// TIA Portal project "HydroelectricDam Project" (V15)

(* hardware
DEVICE "S71500/ET200MP station_1"  S7-1500 station
   slot 0: "Rail_0"  Rack  6ES7 590-1***0-0AA0
   slot 1: "PLC_1"  CPU 1511-1 PN  6ES7 511-1AK00-0AB0  V1.8
      slot 3: "CPU display_1"  6ES7591-1AA00-0AA0
DEVICE "PC-System_1"  SIMATIC PC station
   slot 0: "SIMATIC PC station"  Rail  SIMATIC PC-Station  V1.0
      slot 125: "Stationmanager"  Station_Manager  V6.0.4
   slot 1: "HMI_RT_1"  WinCC RT Advanced  6AV2 104-0xxxx-xxxx  15.0.0.0
      slot 33792: "Host interface"  Host interface
   slot 2: "IE general_1"  IE General  IE_CP  V8.2.0
*)

// ===== PLC "PLC_1"  CPU 1511-1 PN =====

VAR_GLOBAL   // PLC tag table "Default tag table"
   "Brake_Out" AT %M0.0 : Bool;
   "Baffle_Out" AT %MW18 : Int;
   "RPM_In" AT %MW2 : Int;
   "OilTemp_In" AT %MW4 : Int;
   "Baffle_En" AT %M0.1 : Bool;
   "Current_In" AT %MW6 : Int;
   "OilPumpVFDsp_Out" AT %MW8 : Int;
   "OilPumpVFDen_Out" AT %M0.2 : Bool;
   "OilFlow_In" AT %MW10 : Int;
   "PB_LAD" AT %M0.3 : Bool;
   "ONS" AT %M0.4 : Bool;
   "ProgLang" AT %MW12 : Int;
   "PB_FBD" AT %M0.5 : Bool;
   "PB_SCL" AT %M0.6 : Bool;
   "PB_STL" AT %M0.7 : Bool;
   "ONS1" AT %M1.0 : Bool;
   "ONS2" AT %M1.1 : Bool;
   "ONS3" AT %M1.2 : Bool;
   "AlarmHorn_Out" AT %M1.3 : Bool;
   "StationInterlock_Out" AT %M1.4 : Bool;
   "OilPump_VFD_Pct" AT %MW14 : Int;
   "Baffle_Pct" AT %MW16 : Int;
   "OilTemp" AT %MW20 : Int;
   "OilFlow" AT %MW22 : Int;
   "RPM" AT %MW24 : Int;
   "Current" AT %MW26 : Int;
   "SimLogicEn" AT %M1.5 : Bool;
   "OilPumpVFD_Off_Pb" AT %M1.6 : Bool;
   "OilPumpVFD_Hand_Pb" AT %M1.7 : Bool;
   "OilPumpVFD_Auto_Pb" AT %M30.0 : Bool;
   "Brake_Off_Pb" AT %M30.1 : Bool;
   "Brake_hand_Pb" AT %M30.2 : Bool;
   "Brake_Auto_Pb" AT %M30.3 : Bool;
   "Brake_HOA" AT %MW32 : Int;
   "AlarmHorn_Off_Pb" AT %M30.4 : Bool;
   "AlarmHorn_Hand_Pb" AT %M30.5 : Bool;
   "AlarmHorn_Auto_Pb" AT %M30.6 : Bool;
   "AlarmHorn_HOA" AT %MW34 : Int;
   "StationInterlock_Off_Pb" AT %M30.7 : Bool;
   "StationInterlock_Hand_Pb" AT %M31.0 : Bool;
   "StationInterlock_Auto_Pb" AT %M31.1 : Bool;
   "StationInterlock_HOA" AT %MW36 : Int;
   "OilPumpVFD_Ctrl" AT %M31.2 : Bool;
   "Brake_Ctrl" AT %M31.3 : Bool;
   "Alarm_Horn_Ctrl" AT %M31.4 : Bool;
   "StationInterlock_Ctrl" AT %M31.5 : Bool;
   "AlarmReset" AT %M31.6 : Bool;
   "AlarmSilence" AT %M31.7 : Bool;
   "OilLowFlowAlarm" AT %M42.0 : Bool;
   "OilLowFlowNotify" AT %M42.1 : Bool;
   "OilLowFlow_Sp" AT %MW44 : Int;
   "OvercurrentDelaySpt" AT %MW46 : Int;
   "Overcurrent_Sp" AT %MW48 : Int;
   "OvercurrentAlarm" AT %M42.2 : Bool;
   "OvercurrentNotify" AT %M42.3 : Bool;
   "HighOilTempDelaySpt" AT %MW50 : Int;
   "HighOilTemp_Sp" AT %MW52 : Int;
   "HighOilTempAlarm" AT %M42.4 : Bool;
   "HighOiltempNotify" AT %M42.5 : Bool;
   "RotorOverpeedDelaySpt" AT %MW54 : Int;
   "RotorSpeed_Sp" AT %MW56 : Int;
   "RotorOverspeedAlarm" AT %M42.6 : Bool;
   "RotorOverspeedNotify" AT %M42.7 : Bool;
   "OilFlowHighDelaySpt" AT %MW58 : Int;
   "OilFlowhigh_Sp" AT %MW62 : Int;
   "OilFlowHighAlarm" AT %M43.0 : Bool;
   "OilFlowHighNotify" AT %M43.1 : Bool;
   "BrakeFailureDelaySpt" AT %MW64 : Int;
   "BrakeFailureAlarm" AT %M43.2 : Bool;
   "BrakeFailureNotify" AT %M43.3 : Bool;
   "Estop" AT %M43.4 : Bool;
   "EstopAlarm" AT %M43.5 : Bool;
   "EstopNotify" AT %M43.6 : Bool;
   "OilLowFlowDelaySpt" AT %MW60 : Int;
   "Tag_1" AT %T1 : Timer;
   "WarmupMode" AT %M38.0 : Bool;
   "StabilizeMode" AT %M38.1 : Bool;
   "GenerationMode" AT %M38.2 : Bool;
   "CooldownMode" AT %M38.3 : Bool;
   "FaultMode" AT %M38.4 : Bool;
   "IdleMode" AT %M38.5 : Bool;
   "Baffle_HOA" AT %MW40 : Int;
   "Baffle_Ctrl" AT %M38.6 : Bool;
   "WarmupRPM" AT %MW66 : Int;
   "RPM_sp" AT %MW68 : Int;
   "VFD_sp" AT %MW70 : Int;
   "WarmupOilTemp" AT %MW74 : Int;
   "WarmupOilDelay_Sp" AT %MW76 : Int;
   "WarmupTransition" AT %M38.7 : Bool;
   "BafflePID_In" AT %MW78 : Int;
   "BafflePID_Sp" AT %MW80 : Int;
   "StabilizeKW_Sp" AT %MW82 : Int;
   "StabilizeTransition" AT %M39.0 : Bool;
   "StabilizeDelay_Sp" AT %MW86 : Int;
   "SystemStart_PB" AT %M39.1 : Bool;
   "StartSequenceBit" AT %M39.2 : Bool;
   "GenerationTransition" AT %M39.3 : Bool;
   "SystemStop_PB" AT %M39.4 : Bool;
   "CooldownRPM" AT %MW84 : Int;
   "CooldownDelay_Sp" AT %MW88 : Int;
   "CooldownTransition" AT %M39.5 : Bool;
   "CooldownOiltemp_Sp" AT %MW90 : Int;
   "SequenceRunning" AT %M39.6 : Bool;
   "InitializeSequence" AT %M39.7 : Bool;
   "ONS4" AT %M43.7 : Bool;
   "HOFOverrideVFD_Sp" AT %MW92 : Int;
   "Bafflehand_Pb" AT %M94.0 : Bool;
   "BaffleAuto_Pb" AT %M94.1 : Bool;
   "BaffleManual" AT %M94.2 : Bool;
   "BaffleOff_Pb" AT %M94.3 : Bool;
   "Baffle_Manual_Sp" AT %MD96 : Real;
   "ONS8" AT %M94.5 : Bool;
   "ONS5" AT %M94.6 : Bool;
   "ONS6" AT %M94.7 : Bool;
   "ONS7" AT %M95.0 : Bool;
   "ONS9" AT %M95.1 : Bool;
   "VFDhand_Pb" AT %M95.2 : Bool;
   "VFDOff_Pb" AT %M95.3 : Bool;
   "VFDAuto_Pb" AT %M95.4 : Bool;
   "ONS10" AT %M95.5 : Bool;
   "ONS11" AT %M95.6 : Bool;
   "ONS12" AT %M95.7 : Bool;
   "VFD_HOA" AT %MW106 : Int;
   "VFD_Manual_Sp" AT %MD102 : Real;
   "ONS13" AT %M101.0 : Bool;
   "ONS14" AT %M101.1 : Bool;
   "VFDManual" AT %M101.2 : Bool;
   "BafflePID_On" AT %M101.3 : Bool;
   "OilPumpVFD_On" AT %M101.4 : Bool;
   "Full_Auto_Bit" AT %M100.0 : Bool;
   "Warmup_VFD_Pct" AT %MW110 : Int;
   "HM_Minutes" AT %MW28 : Int;
   "Reset_HourMeter_Pb" AT %M72.1 : Bool;
   "HM_Hours" AT %MW108 : Int;
   "HM_Days" AT %MW112 : Int;
   "ModeInt" AT %MW114 : Int;
   "BFAlarm_int" AT %MW116 : Int;
   "ESAlarm_int" AT %MW118 : Int;
   "ROSAlarm_int" AT %MW120 : Int;
   "OvercurrentAlarm_int" AT %MW122 : Int;
   "OFHAlarm_int" AT %MW124 : Int;
   "OFLAlarm_int" AT %MW126 : Int;
   "HOTAlarm_int" AT %MW128 : Int;
   "OS1" AT %M72.0 : Bool;
   "OS2" AT %M72.2 : Bool;
   "OS3" AT %M72.3 : Bool;
   "OS4" AT %M72.4 : Bool;
   "OS5" AT %M72.5 : Bool;
   "OS6" AT %M72.6 : Bool;
   "OS7" AT %M72.7 : Bool;
   "OS8" AT %M73.0 : Bool;
   "OS9" AT %M73.1 : Bool;
   "OS10" AT %M73.2 : Bool;
   "OS11" AT %M73.3 : Bool;
   "OS12" AT %M73.4 : Bool;
   "OS13" AT %M73.5 : Bool;
   "OS14" AT %M73.6 : Bool;
END_VAR

DATA_BLOCK "SimLogic_DB"   // DB1
{ S7_Optimized_Access := 'TRUE' }
VERSION : 0.1
// stored: InstanceOfName SimLogic
"SimLogic"
BEGIN
END_DATA_BLOCK

DATA_BLOCK "IO_LAD_DB"   // DB2
{ S7_Optimized_Access := 'TRUE' }
VERSION : 0.1
// stored: InstanceOfName IO_LAD
"IO_LAD"
BEGIN
END_DATA_BLOCK

DATA_BLOCK "IO_FBD_DB"   // DB4
{ S7_Optimized_Access := 'TRUE' }
VERSION : 0.1
// stored: InstanceOfName IO_FBD
"IO_FBD"
BEGIN
END_DATA_BLOCK

DATA_BLOCK "IO_SCL_DB"   // DB5
{ S7_Optimized_Access := 'TRUE' }
VERSION : 0.1
// stored: InstanceOfName IO_SCL
"IO_SCL"
BEGIN
END_DATA_BLOCK

DATA_BLOCK "IO_STL_DB"   // DB6
{ S7_Optimized_Access := 'TRUE' }
VERSION : 0.1
// stored: InstanceOfName IO_STL
"IO_STL"
BEGIN
END_DATA_BLOCK

DATA_BLOCK "ALARMS_LAD_DB"   // DB7
{ S7_Optimized_Access := 'TRUE' }
VERSION : 0.1
// stored: InstanceOfName ALARMS_LAD
"ALARMS_LAD"
BEGIN
END_DATA_BLOCK

DATA_BLOCK "ALARMS_FBD_DB"   // DB8
{ S7_Optimized_Access := 'TRUE' }
VERSION : 0.1
// stored: InstanceOfName ALARMS_FBD
"ALARMS_FBD"
BEGIN
END_DATA_BLOCK

DATA_BLOCK "ALARMS_SCL_DB"   // DB9
{ S7_Optimized_Access := 'TRUE' }
VERSION : 0.1
// stored: InstanceOfName ALARMS_SCL
"ALARMS_SCL"
BEGIN
END_DATA_BLOCK

DATA_BLOCK "ALARMS_STL_DB"   // DB10
{ S7_Optimized_Access := 'TRUE' }
VERSION : 0.1
// stored: InstanceOfName ALARMS_STL
"ALARMS_STL"
BEGIN
END_DATA_BLOCK

DATA_BLOCK "HOA_LAD_DB"   // DB11
{ S7_Optimized_Access := 'TRUE' }
VERSION : 0.1
// stored: InstanceOfName HOA_LAD
"HOA_LAD"
BEGIN
END_DATA_BLOCK

DATA_BLOCK "HOA_FBD_DB"   // DB12
{ S7_Optimized_Access := 'TRUE' }
VERSION : 0.1
// stored: InstanceOfName HOA_FBD
"HOA_FBD"
BEGIN
END_DATA_BLOCK

DATA_BLOCK "HOA_SCL_DB"   // DB13
{ S7_Optimized_Access := 'TRUE' }
VERSION : 0.1
// stored: InstanceOfName HOA_SCL
"HOA_SCL"
BEGIN
END_DATA_BLOCK

DATA_BLOCK "HOA_STL_DB"   // DB14
{ S7_Optimized_Access := 'TRUE' }
VERSION : 0.1
// stored: InstanceOfName HOA_STL
"HOA_STL"
BEGIN
END_DATA_BLOCK

DATA_BLOCK "MODES_LAD_DB"   // DB29
{ S7_Optimized_Access := 'TRUE' }
VERSION : 0.1
// stored: InstanceOfName MODES_LAD
"MODES_LAD"
BEGIN
END_DATA_BLOCK

DATA_BLOCK "MODES_FBD_DB"   // DB33
{ S7_Optimized_Access := 'TRUE' }
VERSION : 0.1
// stored: InstanceOfName MODES_FBD
"MODES_FBD"
BEGIN
END_DATA_BLOCK

DATA_BLOCK "MODES_SCL_DB"   // DB44
{ S7_Optimized_Access := 'TRUE' }
VERSION : 0.1
// stored: InstanceOfName MODES_SCL
"MODES_SCL"
BEGIN
END_DATA_BLOCK

DATA_BLOCK "MODES_STL_DB"   // DB45
{ S7_Optimized_Access := 'TRUE' }
VERSION : 0.1
// stored: InstanceOfName MODES_STL
"MODES_STL"
BEGIN
END_DATA_BLOCK

DATA_BLOCK "SEQUENCE_DB"   // DB58
{ S7_Optimized_Access := 'TRUE' }
VERSION : 0.1
// stored: InstanceOfName SEQUENCE
"SEQUENCE"
BEGIN
END_DATA_BLOCK

DATA_BLOCK "HOURMETER_LAD_DB"   // DB63
{ S7_Optimized_Access := 'TRUE' }
VERSION : 0.1
// stored: InstanceOfName HOURMETER_LAD
"HOURMETER_LAD"
BEGIN
END_DATA_BLOCK

DATA_BLOCK "HOURMETER_FBD_DB"   // DB64
{ S7_Optimized_Access := 'TRUE' }
VERSION : 0.1
// stored: InstanceOfName HOURMETER_FBD
"HOURMETER_FBD"
BEGIN
END_DATA_BLOCK

DATA_BLOCK "HOURMETER_SCL_DB"   // DB65
{ S7_Optimized_Access := 'TRUE' }
VERSION : 0.1
// stored: InstanceOfName HOURMETER_SCL
"HOURMETER_SCL"
BEGIN
END_DATA_BLOCK

DATA_BLOCK "HOURMETER_STL_DB"   // DB66
{ S7_Optimized_Access := 'TRUE' }
VERSION : 0.1
// stored: InstanceOfName HOURMETER_STL
"HOURMETER_STL"
BEGIN
END_DATA_BLOCK

// folder: System blocks/Program resources

DATA_BLOCK "IEC_Timer_0_DB_25"   // DB3
{ S7_Optimized_Access := 'TRUE' }
AUTHOR : Simatic
FAMILY : IEC
NAME : IEC_TMR
VERSION : 1.0
// stored: InstanceOfName IEC_TIMER
"IEC_TIMER"
BEGIN
END_DATA_BLOCK

DATA_BLOCK "IEC_Timer_0_DB_1"   // DB15
{ S7_Optimized_Access := 'TRUE' }
AUTHOR : Simatic
FAMILY : IEC
NAME : IEC_TMR
VERSION : 1.0
// stored: InstanceOfName IEC_TIMER
"IEC_TIMER"
BEGIN
END_DATA_BLOCK

DATA_BLOCK "IEC_Timer_0_DB_2"   // DB16
{ S7_Optimized_Access := 'TRUE' }
AUTHOR : Simatic
FAMILY : IEC
NAME : IEC_TMR
VERSION : 1.0
// stored: InstanceOfName IEC_TIMER
"IEC_TIMER"
BEGIN
END_DATA_BLOCK

DATA_BLOCK "IEC_Timer_0_DB"   // DB17
{ S7_Optimized_Access := 'TRUE' }
AUTHOR : Simatic
FAMILY : IEC
NAME : IEC_TMR
VERSION : 1.0
// stored: InstanceOfName IEC_TIMER
"IEC_TIMER"
BEGIN
END_DATA_BLOCK

DATA_BLOCK "IEC_Timer_0_DB_3"   // DB18
{ S7_Optimized_Access := 'TRUE' }
AUTHOR : Simatic
FAMILY : IEC
NAME : IEC_TMR
VERSION : 1.0
// stored: InstanceOfName IEC_TIMER
"IEC_TIMER"
BEGIN
END_DATA_BLOCK

DATA_BLOCK "IEC_Timer_0_DB_4"   // DB19
{ S7_Optimized_Access := 'TRUE' }
AUTHOR : Simatic
FAMILY : IEC
NAME : IEC_TMR
VERSION : 1.0
// stored: InstanceOfName IEC_TIMER
"IEC_TIMER"
BEGIN
END_DATA_BLOCK

DATA_BLOCK "IEC_Timer_0_DB_5"   // DB20
{ S7_Optimized_Access := 'TRUE' }
AUTHOR : Simatic
FAMILY : IEC
NAME : IEC_TMR
VERSION : 1.0
// stored: InstanceOfName IEC_TIMER
"IEC_TIMER"
BEGIN
END_DATA_BLOCK

DATA_BLOCK "IEC_Timer_0_DB_6"   // DB21
{ S7_Optimized_Access := 'TRUE' }
AUTHOR : Simatic
FAMILY : IEC
NAME : IEC_TMR
VERSION : 1.0
// stored: InstanceOfName IEC_TIMER
"IEC_TIMER"
BEGIN
END_DATA_BLOCK

DATA_BLOCK "IEC_Timer_0_DB_7"   // DB22
{ S7_Optimized_Access := 'TRUE' }
AUTHOR : Simatic
FAMILY : IEC
NAME : IEC_TMR
VERSION : 1.0
// stored: InstanceOfName IEC_TIMER
"IEC_TIMER"
BEGIN
END_DATA_BLOCK

DATA_BLOCK "IEC_Timer_0_DB_8"   // DB23
{ S7_Optimized_Access := 'TRUE' }
AUTHOR : Simatic
FAMILY : IEC
NAME : IEC_TMR
VERSION : 1.0
// stored: InstanceOfName IEC_TIMER
"IEC_TIMER"
BEGIN
END_DATA_BLOCK

DATA_BLOCK "IEC_Timer_0_DB_9"   // DB24
{ S7_Optimized_Access := 'TRUE' }
AUTHOR : Simatic
FAMILY : IEC
NAME : IEC_TMR
VERSION : 1.0
// stored: InstanceOfName IEC_TIMER
"IEC_TIMER"
BEGIN
END_DATA_BLOCK

DATA_BLOCK "IEC_Timer_0_DB_10"   // DB25
{ S7_Optimized_Access := 'TRUE' }
AUTHOR : Simatic
FAMILY : IEC
NAME : IEC_TMR
VERSION : 1.0
// stored: InstanceOfName IEC_TIMER
"IEC_TIMER"
BEGIN
END_DATA_BLOCK

DATA_BLOCK "IEC_Timer_0_DB_11"   // DB26
{ S7_Optimized_Access := 'TRUE' }
AUTHOR : Simatic
FAMILY : IEC
NAME : IEC_TMR
VERSION : 1.0
// stored: InstanceOfName IEC_TIMER
"IEC_TIMER"
BEGIN
END_DATA_BLOCK

DATA_BLOCK "IEC_Timer_0_DB_12"   // DB27
{ S7_Optimized_Access := 'TRUE' }
AUTHOR : Simatic
FAMILY : IEC
NAME : IEC_TMR
VERSION : 1.0
// stored: InstanceOfName IEC_TIMER
"IEC_TIMER"
BEGIN
END_DATA_BLOCK

DATA_BLOCK "IEC_Timer_0_DB_13"   // DB28
{ S7_Optimized_Access := 'TRUE' }
AUTHOR : Simatic
FAMILY : IEC
NAME : IEC_TMR
VERSION : 1.0
// stored: InstanceOfName IEC_TIMER
"IEC_TIMER"
BEGIN
END_DATA_BLOCK

DATA_BLOCK "IEC_Timer_0_DB_15"   // DB30
{ S7_Optimized_Access := 'TRUE' }
AUTHOR : Simatic
FAMILY : IEC
NAME : IEC_TMR
VERSION : 1.0
// stored: InstanceOfName IEC_TIMER
"IEC_TIMER"
BEGIN
END_DATA_BLOCK

DATA_BLOCK "IEC_Timer_0_DB_16"   // DB31
{ S7_Optimized_Access := 'TRUE' }
AUTHOR : Simatic
FAMILY : IEC
NAME : IEC_TMR
VERSION : 1.0
// stored: InstanceOfName IEC_TIMER
"IEC_TIMER"
BEGIN
END_DATA_BLOCK

DATA_BLOCK "IEC_Timer_0_DB_17"   // DB32
{ S7_Optimized_Access := 'TRUE' }
AUTHOR : Simatic
FAMILY : IEC
NAME : IEC_TMR
VERSION : 1.0
// stored: InstanceOfName IEC_TIMER
"IEC_TIMER"
BEGIN
END_DATA_BLOCK

DATA_BLOCK "IEC_Timer_0_DB_19"   // DB34
{ S7_Optimized_Access := 'TRUE' }
AUTHOR : Simatic
FAMILY : IEC
NAME : IEC_TMR
VERSION : 1.0
// stored: InstanceOfName IEC_TIMER
"IEC_TIMER"
BEGIN
END_DATA_BLOCK

DATA_BLOCK "IEC_Timer_0_DB_20"   // DB35
{ S7_Optimized_Access := 'TRUE' }
AUTHOR : Simatic
FAMILY : IEC
NAME : IEC_TMR
VERSION : 1.0
// stored: InstanceOfName IEC_TIMER
"IEC_TIMER"
BEGIN
END_DATA_BLOCK

DATA_BLOCK "IEC_Timer_0_DB_21"   // DB36
{ S7_Optimized_Access := 'TRUE' }
AUTHOR : Simatic
FAMILY : IEC
NAME : IEC_TMR
VERSION : 1.0
// stored: InstanceOfName IEC_TIMER
"IEC_TIMER"
BEGIN
END_DATA_BLOCK

DATA_BLOCK "IEC_Timer_0_DB_22"   // DB37
{ S7_Optimized_Access := 'TRUE' }
AUTHOR : Simatic
FAMILY : IEC
NAME : IEC_TMR
VERSION : 1.0
// stored: InstanceOfName IEC_TIMER
"IEC_TIMER"
BEGIN
END_DATA_BLOCK

DATA_BLOCK "IEC_Timer_0_DB_23"   // DB38
{ S7_Optimized_Access := 'TRUE' }
AUTHOR : Simatic
FAMILY : IEC
NAME : IEC_TMR
VERSION : 1.0
// stored: InstanceOfName IEC_TIMER
"IEC_TIMER"
BEGIN
END_DATA_BLOCK

DATA_BLOCK "IEC_Timer_0_DB_24"   // DB39
{ S7_Optimized_Access := 'TRUE' }
AUTHOR : Simatic
FAMILY : IEC
NAME : IEC_TMR
VERSION : 1.0
// stored: InstanceOfName IEC_TIMER
"IEC_TIMER"
BEGIN
END_DATA_BLOCK

DATA_BLOCK "IEC_Timer_0_DB_26"   // DB40
{ S7_Optimized_Access := 'TRUE' }
AUTHOR : Simatic
FAMILY : IEC
NAME : IEC_TMR
VERSION : 1.0
// stored: InstanceOfName IEC_TIMER
"IEC_TIMER"
BEGIN
END_DATA_BLOCK

DATA_BLOCK "IEC_Timer_0_DB_27"   // DB41
{ S7_Optimized_Access := 'TRUE' }
AUTHOR : Simatic
FAMILY : IEC
NAME : IEC_TMR
VERSION : 1.0
// stored: InstanceOfName IEC_TIMER
"IEC_TIMER"
BEGIN
END_DATA_BLOCK

DATA_BLOCK "IEC_Timer_1_DB"   // DB43
{ S7_Optimized_Access := 'TRUE' }
AUTHOR : Simatic
FAMILY : IEC
NAME : IEC_TMR
VERSION : 1.0
// stored: InstanceOfName IEC_TIMER
"IEC_TIMER"
BEGIN
END_DATA_BLOCK

DATA_BLOCK "IEC_Timer_0_DB_14"   // DB46
{ S7_Optimized_Access := 'TRUE' }
AUTHOR : Simatic
FAMILY : IEC
NAME : IEC_TMR
VERSION : 1.0
// stored: InstanceOfName IEC_TIMER
"IEC_TIMER"
BEGIN
END_DATA_BLOCK

DATA_BLOCK "IEC_Timer_0_DB_18"   // DB47
{ S7_Optimized_Access := 'TRUE' }
AUTHOR : Simatic
FAMILY : IEC
NAME : IEC_TMR
VERSION : 1.0
// stored: InstanceOfName IEC_TIMER
"IEC_TIMER"
BEGIN
END_DATA_BLOCK

DATA_BLOCK "IEC_Timer_0_DB_28"   // DB48
{ S7_Optimized_Access := 'TRUE' }
AUTHOR : Simatic
FAMILY : IEC
NAME : IEC_TMR
VERSION : 1.0
// stored: InstanceOfName IEC_TIMER
"IEC_TIMER"
BEGIN
END_DATA_BLOCK

DATA_BLOCK "IEC_Timer_0_DB_29"   // DB49
{ S7_Optimized_Access := 'TRUE' }
AUTHOR : Simatic
FAMILY : IEC
NAME : IEC_TMR
VERSION : 1.0
// stored: InstanceOfName IEC_TIMER
"IEC_TIMER"
BEGIN
END_DATA_BLOCK

DATA_BLOCK "IEC_Timer_0_DB_30"   // DB50
{ S7_Optimized_Access := 'TRUE' }
AUTHOR : Simatic
FAMILY : IEC
NAME : IEC_TMR
VERSION : 1.0
// stored: InstanceOfName IEC_TIMER
"IEC_TIMER"
BEGIN
END_DATA_BLOCK

DATA_BLOCK "IEC_Timer_0_DB_31"   // DB51
{ S7_Optimized_Access := 'TRUE' }
AUTHOR : Simatic
FAMILY : IEC
NAME : IEC_TMR
VERSION : 1.0
// stored: InstanceOfName IEC_TIMER
"IEC_TIMER"
BEGIN
END_DATA_BLOCK

DATA_BLOCK "IEC_Timer_0_DB_32"   // DB52
{ S7_Optimized_Access := 'TRUE' }
AUTHOR : Simatic
FAMILY : IEC
NAME : IEC_TMR
VERSION : 1.0
// stored: InstanceOfName IEC_TIMER
"IEC_TIMER"
BEGIN
END_DATA_BLOCK

DATA_BLOCK "IEC_Timer_0_DB_33"   // DB53
{ S7_Optimized_Access := 'TRUE' }
AUTHOR : Simatic
FAMILY : IEC
NAME : IEC_TMR
VERSION : 1.0
// stored: InstanceOfName IEC_TIMER
"IEC_TIMER"
BEGIN
END_DATA_BLOCK

DATA_BLOCK "IEC_Timer_0_DB_34"   // DB54
{ S7_Optimized_Access := 'TRUE' }
AUTHOR : Simatic
FAMILY : IEC
NAME : IEC_TMR
VERSION : 1.0
// stored: InstanceOfName IEC_TIMER
"IEC_TIMER"
BEGIN
END_DATA_BLOCK

DATA_BLOCK "IEC_Timer_0_DB_35"   // DB55
{ S7_Optimized_Access := 'TRUE' }
AUTHOR : Simatic
FAMILY : IEC
NAME : IEC_TMR
VERSION : 1.0
// stored: InstanceOfName IEC_TIMER
"IEC_TIMER"
BEGIN
END_DATA_BLOCK

DATA_BLOCK "IEC_Timer_0_DB_36"   // DB56
{ S7_Optimized_Access := 'TRUE' }
AUTHOR : Simatic
FAMILY : IEC
NAME : IEC_TMR
VERSION : 1.0
// stored: InstanceOfName IEC_TIMER
"IEC_TIMER"
BEGIN
END_DATA_BLOCK

DATA_BLOCK "IEC_Timer_0_DB_37"   // DB57
{ S7_Optimized_Access := 'TRUE' }
AUTHOR : Simatic
FAMILY : IEC
NAME : IEC_TMR
VERSION : 1.0
// stored: InstanceOfName IEC_TIMER
"IEC_TIMER"
BEGIN
END_DATA_BLOCK

DATA_BLOCK "IEC_Timer_0_DB_38"   // DB67
{ S7_Optimized_Access := 'TRUE' }
AUTHOR : Simatic
FAMILY : IEC
NAME : IEC_TMR
VERSION : 1.0
// stored: InstanceOfName IEC_TIMER
"IEC_TIMER"
BEGIN
END_DATA_BLOCK

DATA_BLOCK "IEC_Counter_0_DB"   // DB68
{ S7_Optimized_Access := 'TRUE' }
AUTHOR : Simatic
FAMILY : IEC
NAME : CNTR
VERSION : 1.0
// stored: InstanceOfName IEC_COUNTER
"IEC_COUNTER"
BEGIN
END_DATA_BLOCK

DATA_BLOCK "IEC_Counter_0_DB_1"   // DB69
{ S7_Optimized_Access := 'TRUE' }
AUTHOR : Simatic
FAMILY : IEC
NAME : CNTR
VERSION : 1.0
// stored: InstanceOfName IEC_COUNTER
"IEC_COUNTER"
BEGIN
END_DATA_BLOCK

DATA_BLOCK "IEC_Counter_0_DB_11"   // DB70
{ S7_Optimized_Access := 'TRUE' }
AUTHOR : Simatic
FAMILY : IEC
NAME : CNTR
VERSION : 1.0
// stored: InstanceOfName IEC_COUNTER
"IEC_COUNTER"
BEGIN
END_DATA_BLOCK

DATA_BLOCK "IEC_Counter_0_DB_3"   // DB71
{ S7_Optimized_Access := 'TRUE' }
AUTHOR : Simatic
FAMILY : IEC
NAME : CNTR
VERSION : 1.0
// stored: InstanceOfName IEC_COUNTER
"IEC_COUNTER"
BEGIN
END_DATA_BLOCK

DATA_BLOCK "IEC_Timer_0_DB_39"   // DB72
{ S7_Optimized_Access := 'TRUE' }
AUTHOR : Simatic
FAMILY : IEC
NAME : IEC_TMR
VERSION : 1.0
// stored: InstanceOfName IEC_TIMER
"IEC_TIMER"
BEGIN
END_DATA_BLOCK

DATA_BLOCK "IEC_Timer_0_DB_40"   // DB73
{ S7_Optimized_Access := 'TRUE' }
AUTHOR : Simatic
FAMILY : IEC
NAME : IEC_TMR
VERSION : 1.0
// stored: InstanceOfName IEC_TIMER
"IEC_TIMER"
BEGIN
END_DATA_BLOCK

DATA_BLOCK "IEC_Counter_0_DB_4"   // DB74
{ S7_Optimized_Access := 'TRUE' }
AUTHOR : Simatic
FAMILY : IEC
NAME : CNTR
VERSION : 1.0
// stored: InstanceOfName IEC_COUNTER
"IEC_COUNTER"
BEGIN
END_DATA_BLOCK

DATA_BLOCK "IEC_Timer_0_DB_41"   // DB75
{ S7_Optimized_Access := 'TRUE' }
AUTHOR : Simatic
FAMILY : IEC
NAME : IEC_TMR
VERSION : 1.0
// stored: InstanceOfName IEC_TIMER
"IEC_TIMER"
BEGIN
END_DATA_BLOCK

DATA_BLOCK "IEC_Timer_0_DB_42"   // DB76
{ S7_Optimized_Access := 'TRUE' }
AUTHOR : Simatic
FAMILY : IEC
NAME : IEC_TMR
VERSION : 1.0
// stored: InstanceOfName IEC_TIMER
"IEC_TIMER"
BEGIN
END_DATA_BLOCK

DATA_BLOCK "IEC_Counter_0_DB_5"   // DB77
{ S7_Optimized_Access := 'TRUE' }
AUTHOR : Simatic
FAMILY : IEC
NAME : CNTR
VERSION : 1.0
// stored: InstanceOfName IEC_COUNTER
"IEC_COUNTER"
BEGIN
END_DATA_BLOCK

DATA_BLOCK "IEC_Counter_0_DB_6"   // DB78
{ S7_Optimized_Access := 'TRUE' }
AUTHOR : Simatic
FAMILY : IEC
NAME : CNTR
VERSION : 1.0
// stored: InstanceOfName IEC_COUNTER
"IEC_COUNTER"
BEGIN
END_DATA_BLOCK

DATA_BLOCK "IEC_Counter_0_DB_7"   // DB79
{ S7_Optimized_Access := 'TRUE' }
AUTHOR : Simatic
FAMILY : IEC
NAME : CNTR
VERSION : 1.0
// stored: InstanceOfName IEC_COUNTER
"IEC_COUNTER"
BEGIN
END_DATA_BLOCK

DATA_BLOCK "IEC_Timer_0_DB_43"   // DB80
{ S7_Optimized_Access := 'TRUE' }
AUTHOR : Simatic
FAMILY : IEC
NAME : IEC_TMR
VERSION : 1.0
// stored: InstanceOfName IEC_TIMER
"IEC_TIMER"
BEGIN
END_DATA_BLOCK

DATA_BLOCK "IEC_Timer_0_DB_44"   // DB81
{ S7_Optimized_Access := 'TRUE' }
AUTHOR : Simatic
FAMILY : IEC
NAME : IEC_TMR
VERSION : 1.0
// stored: InstanceOfName IEC_TIMER
"IEC_TIMER"
BEGIN
END_DATA_BLOCK

DATA_BLOCK "IEC_Counter_0_DB_8"   // DB82
{ S7_Optimized_Access := 'TRUE' }
AUTHOR : Simatic
FAMILY : IEC
NAME : CNTR
VERSION : 1.0
// stored: InstanceOfName IEC_COUNTER
"IEC_COUNTER"
BEGIN
END_DATA_BLOCK

DATA_BLOCK "IEC_Counter_0_DB_9"   // DB83
{ S7_Optimized_Access := 'TRUE' }
AUTHOR : Simatic
FAMILY : IEC
NAME : CNTR
VERSION : 1.0
// stored: InstanceOfName IEC_COUNTER
"IEC_COUNTER"
BEGIN
END_DATA_BLOCK

DATA_BLOCK "IEC_Counter_0_DB_10"   // DB84
{ S7_Optimized_Access := 'TRUE' }
AUTHOR : Simatic
FAMILY : IEC
NAME : CNTR
VERSION : 1.0
// stored: InstanceOfName IEC_COUNTER
"IEC_COUNTER"
BEGIN
END_DATA_BLOCK

DATA_BLOCK "IEC_Timer_0_DB_45"   // DB85
{ S7_Optimized_Access := 'TRUE' }
AUTHOR : Simatic
FAMILY : IEC
NAME : IEC_TMR
VERSION : 1.0
// stored: InstanceOfName IEC_TIMER
"IEC_TIMER"
BEGIN
END_DATA_BLOCK

DATA_BLOCK "IEC_Counter_0_DB_12"   // DB86
{ S7_Optimized_Access := 'TRUE' }
AUTHOR : Simatic
FAMILY : IEC
NAME : CNTR
VERSION : 1.0
// stored: InstanceOfName IEC_COUNTER
"IEC_COUNTER"
BEGIN
END_DATA_BLOCK

// folder: (top level)

FUNCTION_BLOCK "SimLogic"   // FB1, FBD
{ S7_Optimized_Access := 'TRUE' }
VERSION : 0.1
   VAR
      "TO" : Bool;
      rpmv : Int;
      addrpmv : Bool;
      otsp : Int;
      ott : Int;
      TO1 : Bool;
      TO2 : Bool;
      be2 : Int;
      be3 : Int;
      be1 : Int;
      TO3 : Bool;
   END_VAR
   VAR_TEMP
      bf : Int;
      rpmvt : Int;
      bfr : Real;
   END_VAR
BEGIN

REGION Network 1
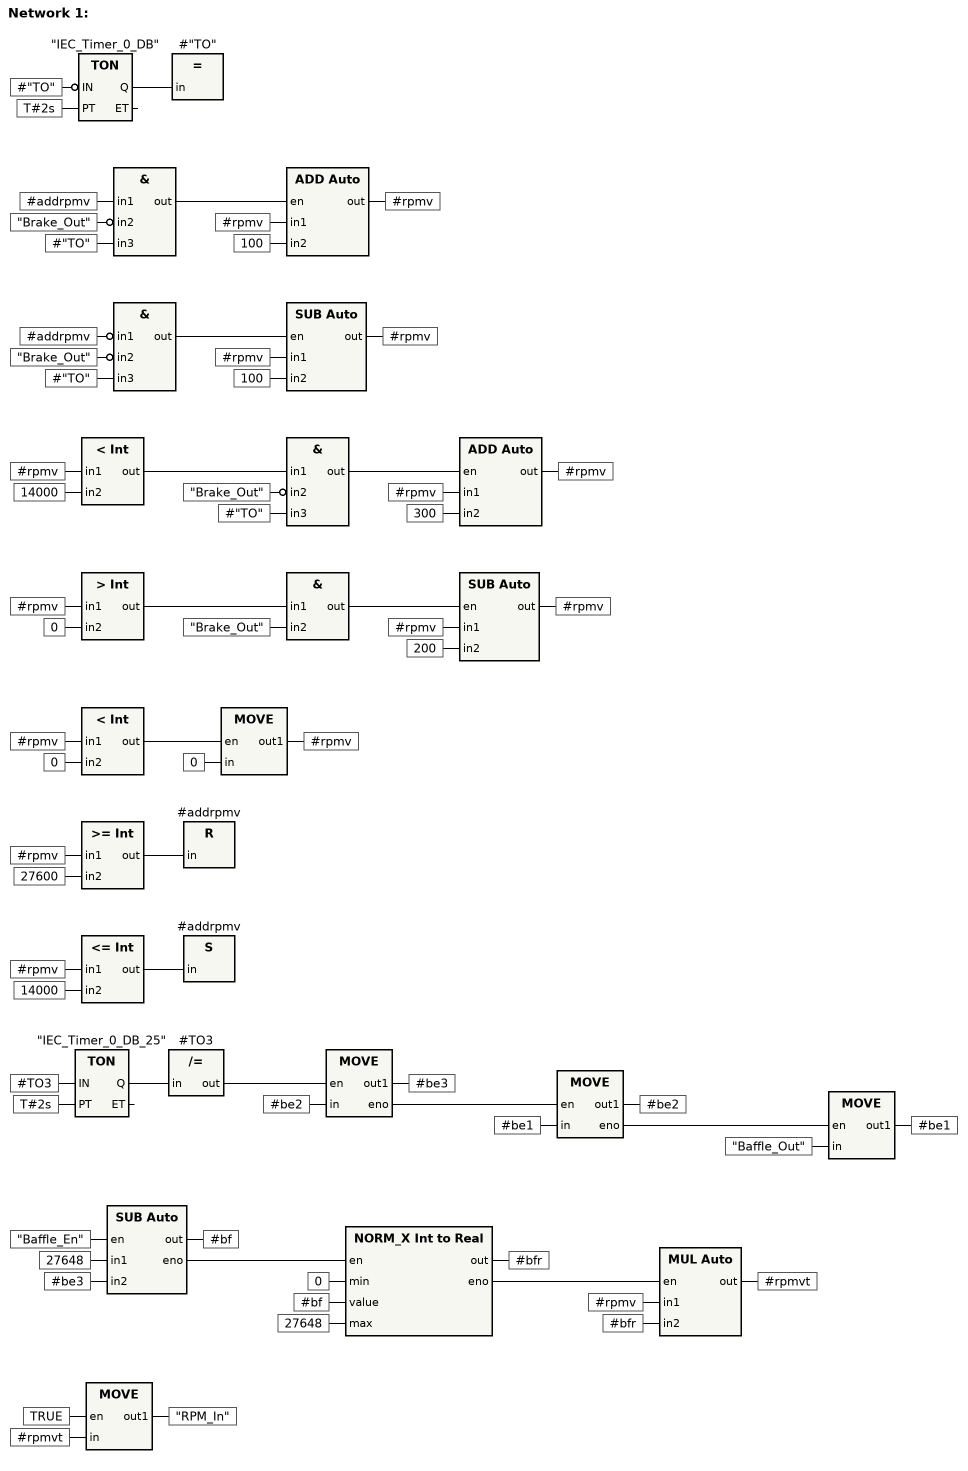
   "IEC_Timer_0_DB".TON(IN := NOT #"TO", PT := T#2s);
   #"TO" := "IEC_Timer_0_DB".Q;
   IF #addrpmv AND NOT "Brake_Out" AND #"TO" THEN #rpmv := #rpmv + 100; END_IF;
   IF NOT #addrpmv AND NOT "Brake_Out" AND #"TO" THEN #rpmv := #rpmv - 100; END_IF;
   IF (#rpmv < 14000) AND NOT "Brake_Out" AND #"TO" THEN #rpmv := #rpmv + 300; END_IF;
   IF (#rpmv > 0) AND "Brake_Out" THEN #rpmv := #rpmv - 200; END_IF;
   IF #rpmv < 0 THEN #rpmv := 0; END_IF;
   IF #rpmv >= 27600 THEN #addrpmv := FALSE; END_IF;
   IF #rpmv <= 14000 THEN #addrpmv := TRUE; END_IF;
   "IEC_Timer_0_DB_25".TON(IN := #TO3, PT := T#2s);
   #TO3 := NOT "IEC_Timer_0_DB_25".Q;
   IF "IEC_Timer_0_DB_25".Q THEN
       #be3 := #be2;
       #be2 := #be1;
       #be1 := "Baffle_Out";
   END_IF;
   IF "Baffle_En" THEN
       #bf := 27648 - #be3;
       #bfr := NORM_X(MIN := 0, VALUE := #bf, MAX := 27648);
       #rpmvt := #rpmv * #bfr;
   END_IF;
   IF TRUE THEN "RPM_In" := #rpmvt; END_IF;
END_REGION

REGION Network 2
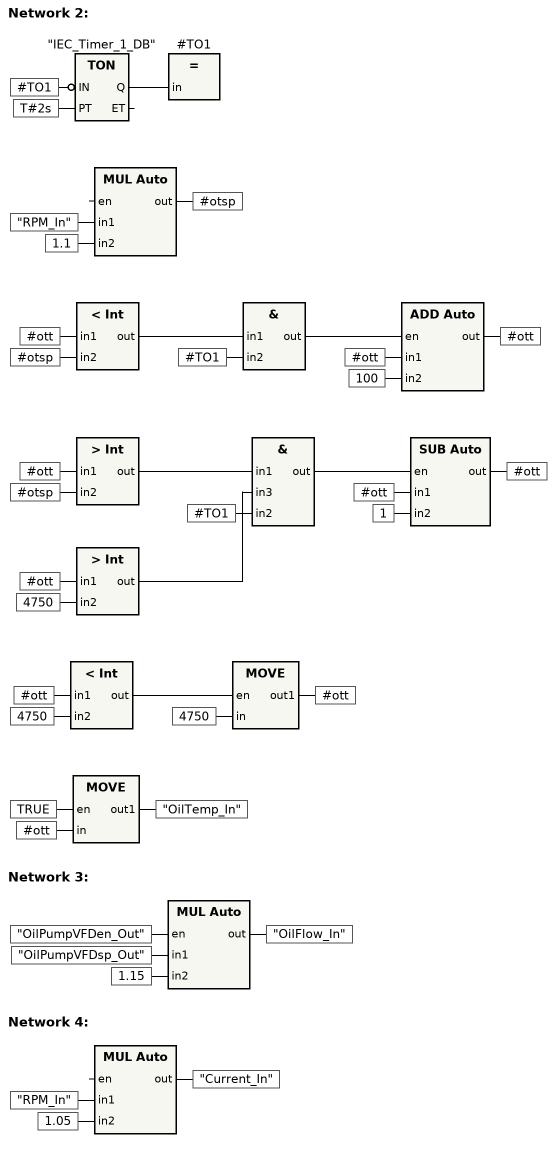
   "IEC_Timer_1_DB".TON(IN := NOT #TO1, PT := T#2s);
   #TO1 := "IEC_Timer_1_DB".Q;
   #otsp := "RPM_In" * 1.1;
   IF (#ott < #otsp) AND #TO1 THEN #ott := #ott + 100; END_IF;
   IF (#ott > #otsp) AND (#ott > 4750) AND #TO1 THEN #ott := #ott - 1; END_IF;
   IF #ott < 4750 THEN #ott := 4750; END_IF;
   IF TRUE THEN "OilTemp_In" := #ott; END_IF;
END_REGION

REGION Network 3
   IF "OilPumpVFDen_Out" THEN "OilFlow_In" := "OilPumpVFDsp_Out" * 1.15; END_IF;
END_REGION

REGION Network 4
   "Current_In" := "RPM_In" * 1.05;
END_REGION
END_FUNCTION_BLOCK

FUNCTION_BLOCK "IO_LAD"   // FB2, LAD
{ S7_Optimized_Access := 'TRUE' }
VERSION : 0.1
BEGIN

REGION Network 1
   // Digital Output
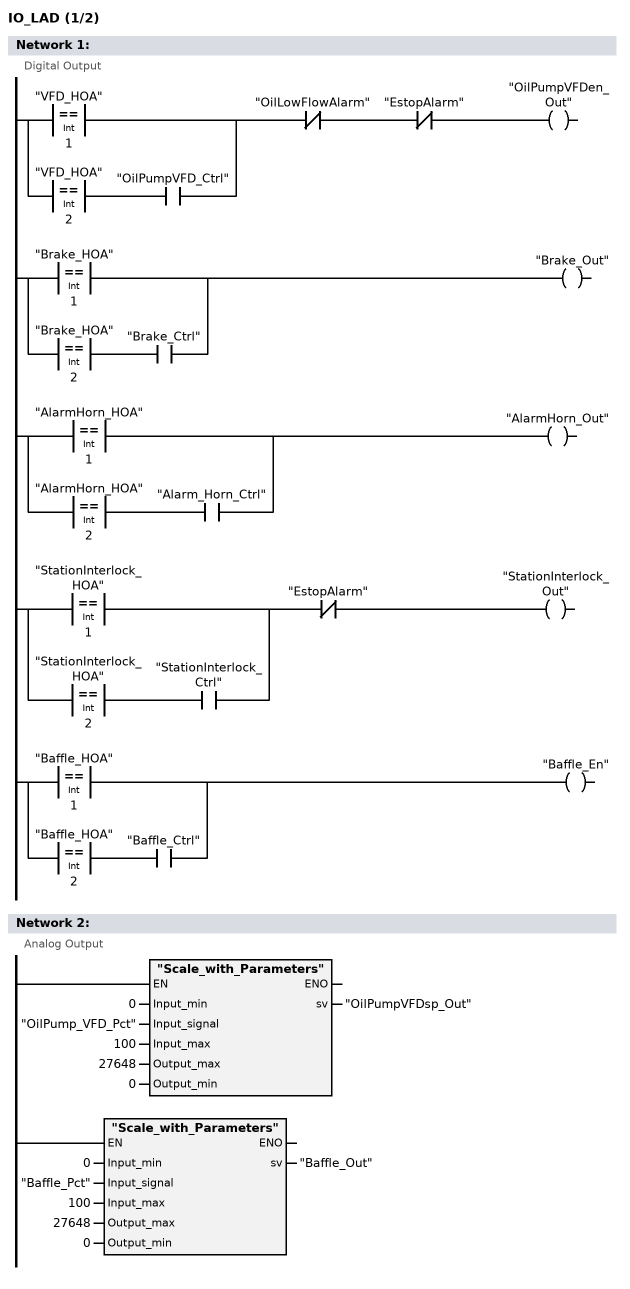
   RUNG wire#powerrail
      { S7_Templates := "SrcType := Int" } EQ_Contact(in1 := "VFD_HOA", in2 := 1)
      wire#w1
      I_Contact( "OilLowFlowAlarm" )
      I_Contact( "EstopAlarm" )
      Coil( "OilPumpVFDen_Out" )
   END_RUNG
   RUNG wire#powerrail
      { S7_Templates := "SrcType := Int" } EQ_Contact(in1 := "VFD_HOA", in2 := 2)
      Contact( "OilPumpVFD_Ctrl" )
   END_RUNG wire#w1
   RUNG wire#powerrail
      { S7_Templates := "SrcType := Int" } EQ_Contact(in1 := "Brake_HOA", in2 := 1)
      wire#w2
      Coil( "Brake_Out" )
   END_RUNG
   RUNG wire#powerrail
      { S7_Templates := "SrcType := Int" } EQ_Contact(in1 := "Brake_HOA", in2 := 2)
      Contact( "Brake_Ctrl" )
   END_RUNG wire#w2
   RUNG wire#powerrail
      { S7_Templates := "SrcType := Int" } EQ_Contact(in1 := "AlarmHorn_HOA", in2 := 1)
      wire#w3
      Coil( "AlarmHorn_Out" )
   END_RUNG
   RUNG wire#powerrail
      { S7_Templates := "SrcType := Int" } EQ_Contact(in1 := "AlarmHorn_HOA", in2 := 2)
      Contact( "Alarm_Horn_Ctrl" )
   END_RUNG wire#w3
   RUNG wire#powerrail
      { S7_Templates := "SrcType := Int" } EQ_Contact(in1 := "StationInterlock_HOA", in2 := 1)
      wire#w4
      I_Contact( "EstopAlarm" )
      Coil( "StationInterlock_Out" )
   END_RUNG
   RUNG wire#powerrail
      { S7_Templates := "SrcType := Int" } EQ_Contact(in1 := "StationInterlock_HOA", in2 := 2)
      Contact( "StationInterlock_Ctrl" )
   END_RUNG wire#w4
   RUNG wire#powerrail
      { S7_Templates := "SrcType := Int" } EQ_Contact(in1 := "Baffle_HOA", in2 := 1)
      wire#w5
      Coil( "Baffle_En" )
   END_RUNG
   RUNG wire#powerrail
      { S7_Templates := "SrcType := Int" } EQ_Contact(in1 := "Baffle_HOA", in2 := 2)
      Contact( "Baffle_Ctrl" )
   END_RUNG wire#w5
   // the same network as SCL:
   "OilPumpVFDen_Out" := (("VFD_HOA" = 1) OR (("VFD_HOA" = 2) AND "OilPumpVFD_Ctrl")) AND NOT "OilLowFlowAlarm" AND NOT "EstopAlarm";
   "Brake_Out" := ("Brake_HOA" = 1) OR (("Brake_HOA" = 2) AND "Brake_Ctrl");
   "AlarmHorn_Out" := ("AlarmHorn_HOA" = 1) OR (("AlarmHorn_HOA" = 2) AND "Alarm_Horn_Ctrl");
   "StationInterlock_Out" := (("StationInterlock_HOA" = 1) OR (("StationInterlock_HOA" = 2) AND "StationInterlock_Ctrl")) AND NOT "EstopAlarm";
   "Baffle_En" := ("Baffle_HOA" = 1) OR (("Baffle_HOA" = 2) AND "Baffle_Ctrl");
END_REGION

REGION Network 2
   // Analog Output
   RUNG wire#powerrail
      "Scale_with_Parameters"(Input_min := 0, Input_signal := "OilPump_VFD_Pct", Input_max := 100, Output_max := 27648, Output_min := 0, sv => "OilPumpVFDsp_Out")
   END_RUNG
   RUNG wire#powerrail
      "Scale_with_Parameters"(Input_min := 0, Input_signal := "Baffle_Pct", Input_max := 100, Output_max := 27648, Output_min := 0, sv => "Baffle_Out")
   END_RUNG
   // the same network as SCL:
   "Scale_with_Parameters"(Input_min := 0,
                           Input_signal := "OilPump_VFD_Pct",
                           Input_max := 100,
                           Output_max := 27648,
                           Output_min := 0,
                           sv => "OilPumpVFDsp_Out");
   "Scale_with_Parameters"(Input_min := 0,
                           Input_signal := "Baffle_Pct",
                           Input_max := 100,
                           Output_max := 27648,
                           Output_min := 0,
                           sv => "Baffle_Out");
END_REGION

REGION Network 3
   // Analog Inputs
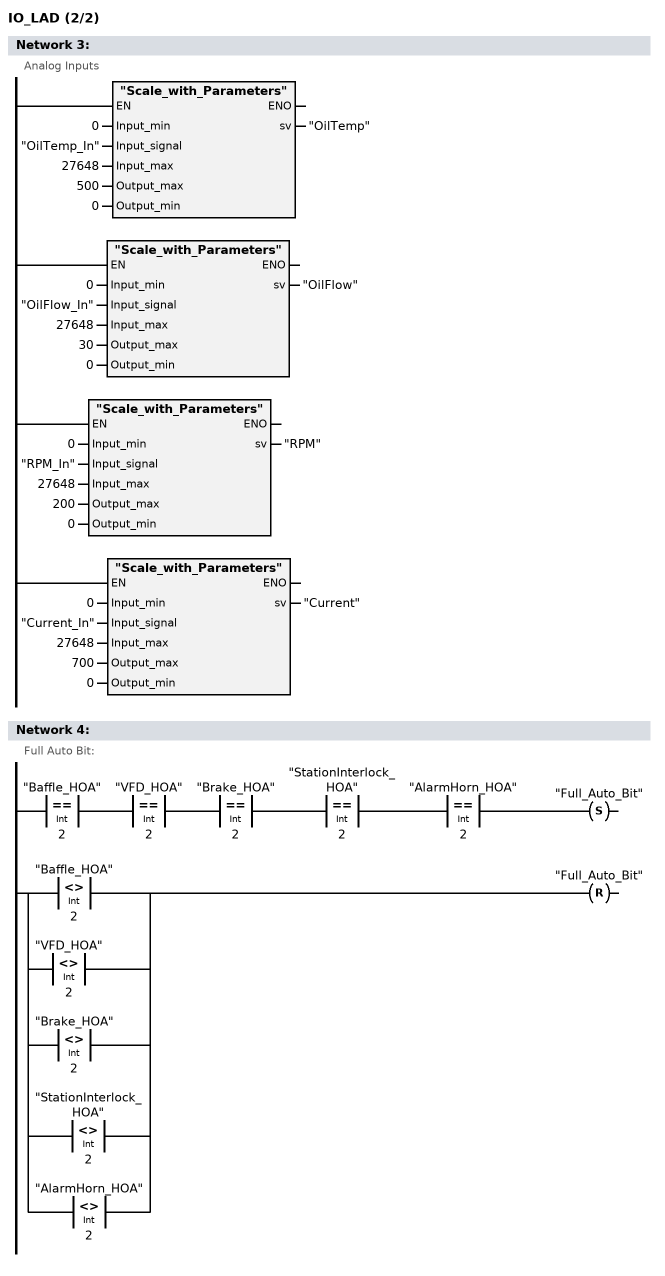
   RUNG wire#powerrail
      "Scale_with_Parameters"(Input_min := 0, Input_signal := "OilTemp_In", Input_max := 27648, Output_max := 500, Output_min := 0, sv => "OilTemp")
   END_RUNG
   RUNG wire#powerrail
      "Scale_with_Parameters"(Input_min := 0, Input_signal := "OilFlow_In", Input_max := 27648, Output_max := 30, Output_min := 0, sv => "OilFlow")
   END_RUNG
   RUNG wire#powerrail
      "Scale_with_Parameters"(Input_min := 0, Input_signal := "RPM_In", Input_max := 27648, Output_max := 200, Output_min := 0, sv => "RPM")
   END_RUNG
   RUNG wire#powerrail
      "Scale_with_Parameters"(Input_min := 0, Input_signal := "Current_In", Input_max := 27648, Output_max := 700, Output_min := 0, sv => "Current")
   END_RUNG
   // the same network as SCL:
   "Scale_with_Parameters"(Input_min := 0,
                           Input_signal := "OilTemp_In",
                           Input_max := 27648,
                           Output_max := 500,
                           Output_min := 0,
                           sv => "OilTemp");
   "Scale_with_Parameters"(Input_min := 0,
                           Input_signal := "OilFlow_In",
                           Input_max := 27648,
                           Output_max := 30,
                           Output_min := 0,
                           sv => "OilFlow");
   "Scale_with_Parameters"(Input_min := 0,
                           Input_signal := "RPM_In",
                           Input_max := 27648,
                           Output_max := 200,
                           Output_min := 0,
                           sv => "RPM");
   "Scale_with_Parameters"(Input_min := 0,
                           Input_signal := "Current_In",
                           Input_max := 27648,
                           Output_max := 700,
                           Output_min := 0,
                           sv => "Current");
END_REGION

REGION Network 4
   // Full Auto Bit:
   RUNG wire#powerrail
      { S7_Templates := "SrcType := Int" } EQ_Contact(in1 := "Baffle_HOA", in2 := 2)
      { S7_Templates := "SrcType := Int" } EQ_Contact(in1 := "VFD_HOA", in2 := 2)
      { S7_Templates := "SrcType := Int" } EQ_Contact(in1 := "Brake_HOA", in2 := 2)
      { S7_Templates := "SrcType := Int" } EQ_Contact(in1 := "StationInterlock_HOA", in2 := 2)
      { S7_Templates := "SrcType := Int" } EQ_Contact(in1 := "AlarmHorn_HOA", in2 := 2)
      S_Coil( "Full_Auto_Bit" )
   END_RUNG
   RUNG wire#powerrail
      { S7_Templates := "SrcType := Int" } NE_Contact(in1 := "Baffle_HOA", in2 := 2)
      wire#w1
      R_Coil( "Full_Auto_Bit" )
   END_RUNG
   RUNG wire#powerrail
      { S7_Templates := "SrcType := Int" } NE_Contact(in1 := "VFD_HOA", in2 := 2)
   END_RUNG wire#w1
   RUNG wire#powerrail
      { S7_Templates := "SrcType := Int" } NE_Contact(in1 := "Brake_HOA", in2 := 2)
   END_RUNG wire#w1
   RUNG wire#powerrail
      { S7_Templates := "SrcType := Int" } NE_Contact(in1 := "StationInterlock_HOA", in2 := 2)
   END_RUNG wire#w1
   RUNG wire#powerrail
      { S7_Templates := "SrcType := Int" } NE_Contact(in1 := "AlarmHorn_HOA", in2 := 2)
   END_RUNG wire#w1
   // the same network as SCL:
   IF ("Baffle_HOA" = 2) AND ("VFD_HOA" = 2) AND ("Brake_HOA" = 2) AND ("StationInterlock_HOA" = 2) AND ("AlarmHorn_HOA" = 2) THEN
       "Full_Auto_Bit" := TRUE;
   END_IF;
   IF ("Baffle_HOA" <> 2) OR ("VFD_HOA" <> 2) OR ("Brake_HOA" <> 2) OR ("StationInterlock_HOA" <> 2) OR ("AlarmHorn_HOA" <> 2) THEN
       "Full_Auto_Bit" := FALSE;
   END_IF;
END_REGION
END_FUNCTION_BLOCK

FUNCTION_BLOCK "IO_FBD"   // FB3, FBD
{ S7_Optimized_Access := 'TRUE' }
VERSION : 0.1
   VAR_TEMP
      tv : Real;
   END_VAR
BEGIN

REGION Network 1
   // Digital outputs:
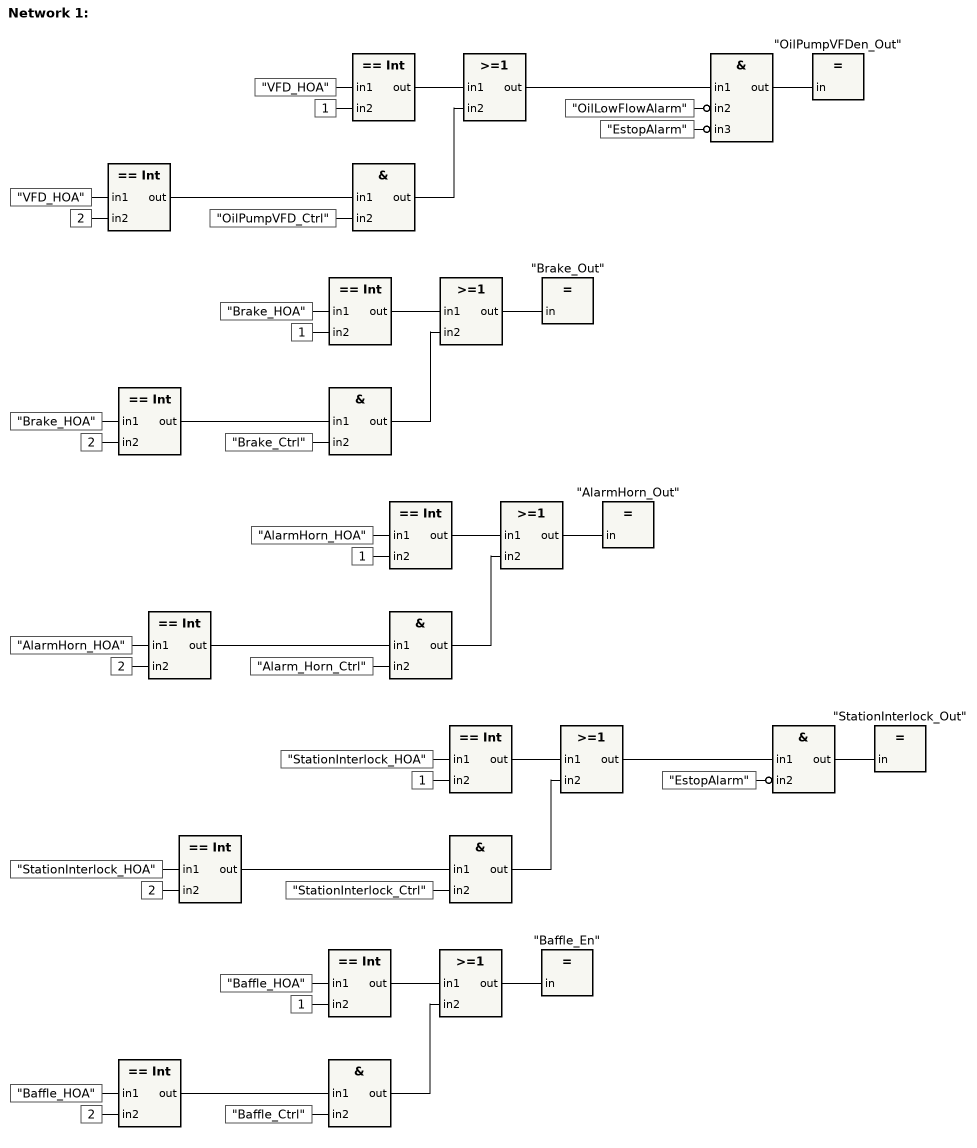
   "OilPumpVFDen_Out" := (("VFD_HOA" = 1) OR (("VFD_HOA" = 2) AND "OilPumpVFD_Ctrl")) AND NOT "OilLowFlowAlarm" AND NOT "EstopAlarm";
   "Brake_Out" := ("Brake_HOA" = 1) OR (("Brake_HOA" = 2) AND "Brake_Ctrl");
   "AlarmHorn_Out" := ("AlarmHorn_HOA" = 1) OR (("AlarmHorn_HOA" = 2) AND "Alarm_Horn_Ctrl");
   "StationInterlock_Out" := (("StationInterlock_HOA" = 1) OR (("StationInterlock_HOA" = 2) AND "StationInterlock_Ctrl")) AND NOT "EstopAlarm";
   "Baffle_En" := ("Baffle_HOA" = 1) OR (("Baffle_HOA" = 2) AND "Baffle_Ctrl");
END_REGION

REGION Network 2
   // Analog output:
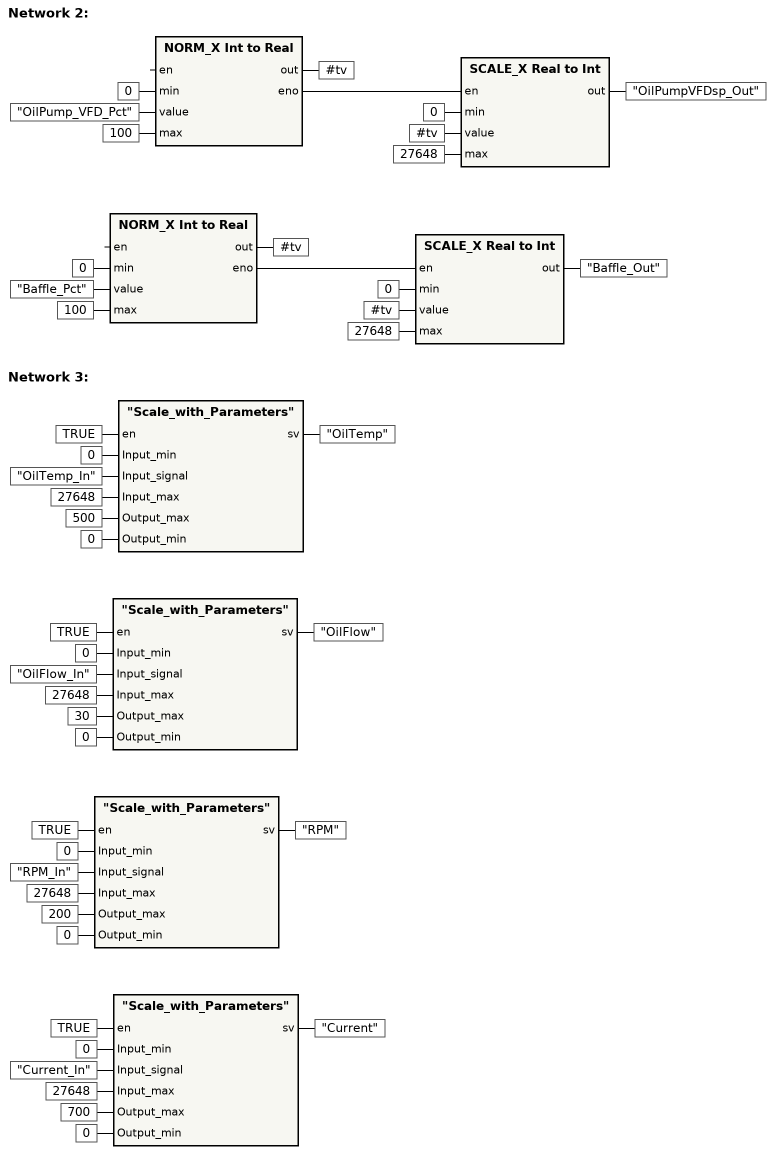
   #tv := NORM_X(MIN := 0, VALUE := "OilPump_VFD_Pct", MAX := 100);
   "OilPumpVFDsp_Out" := SCALE_X(MIN := 0, VALUE := #tv, MAX := 27648);
   #tv := NORM_X(MIN := 0, VALUE := "Baffle_Pct", MAX := 100);
   "Baffle_Out" := SCALE_X(MIN := 0, VALUE := #tv, MAX := 27648);
END_REGION

REGION Network 3
   // Analog Inputs:
   IF TRUE THEN
       "Scale_with_Parameters"(Input_min := 0,
                               Input_signal := "OilTemp_In",
                               Input_max := 27648,
                               Output_max := 500,
                               Output_min := 0,
                               sv => "OilTemp");
       "Scale_with_Parameters"(Input_min := 0,
                               Input_signal := "OilFlow_In",
                               Input_max := 27648,
                               Output_max := 30,
                               Output_min := 0,
                               sv => "OilFlow");
       "Scale_with_Parameters"(Input_min := 0,
                               Input_signal := "RPM_In",
                               Input_max := 27648,
                               Output_max := 200,
                               Output_min := 0,
                               sv => "RPM");
       "Scale_with_Parameters"(Input_min := 0,
                               Input_signal := "Current_In",
                               Input_max := 27648,
                               Output_max := 700,
                               Output_min := 0,
                               sv => "Current");
   END_IF;
END_REGION

REGION Network 4
   // Full Auto Bit
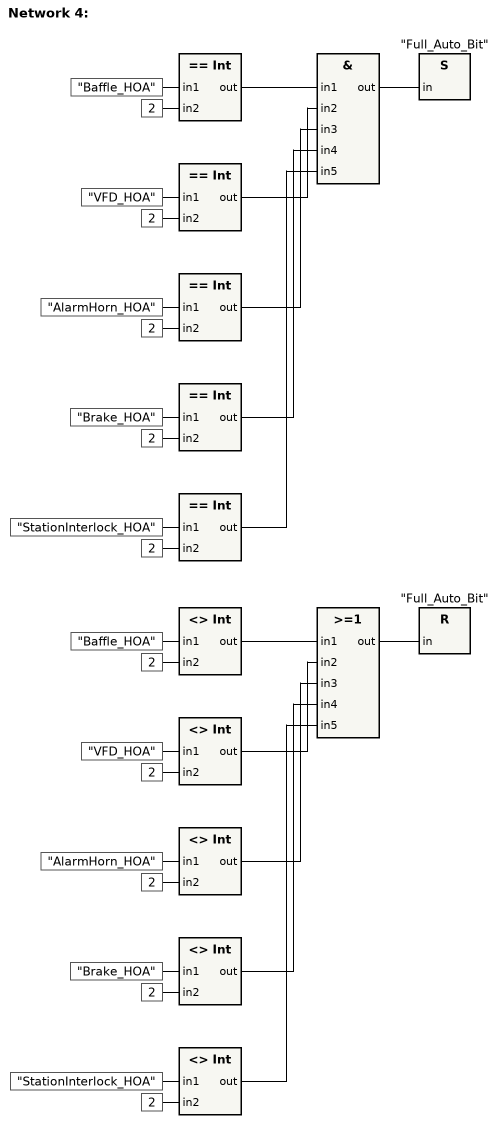
   IF ("Baffle_HOA" = 2) AND ("VFD_HOA" = 2) AND ("AlarmHorn_HOA" = 2) AND ("Brake_HOA" = 2) AND ("StationInterlock_HOA" = 2) THEN
       "Full_Auto_Bit" := TRUE;
   END_IF;
   IF ("Baffle_HOA" <> 2) OR ("VFD_HOA" <> 2) OR ("AlarmHorn_HOA" <> 2) OR ("Brake_HOA" <> 2) OR ("StationInterlock_HOA" <> 2) THEN
       "Full_Auto_Bit" := FALSE;
   END_IF;
END_REGION
END_FUNCTION_BLOCK

FUNCTION_BLOCK "IO_SCL"   // FB4, SCL
{ S7_Optimized_Access := 'TRUE' }
VERSION : 0.1
BEGIN
   //Digital Outputs:

   IF "OilLowFlowAlarm"OR "EstopAlarm" OR  "VFD_HOA" = 0 OR ("VFD_HOA" = 2 AND NOT "OilPumpVFD_Ctrl") THEN
       "OilPumpVFDen_Out" := 0;
   END_IF;

   IF ("VFD_HOA" = 1  OR ("VFD_HOA" = 2 AND "OilPumpVFD_Ctrl")) AND NOT "OilLowFlowAlarm" AND NOT "EstopAlarm" THEN
       "OilPumpVFDen_Out" := 1;
   END_IF;


   IF "Brake_HOA" = 0 OR ("Brake_HOA" = 2 AND NOT "Brake_Ctrl") THEN
       "Brake_Out" := 0;
   END_IF;

   IF "Brake_HOA" = 1 OR ("Brake_HOA" = 2 AND "Brake_Ctrl") THEN
       "Brake_Out" := 1;
   END_IF;



   IF "AlarmHorn_HOA" = 0 OR ("AlarmHorn_HOA" = 2 AND NOT "Alarm_Horn_Ctrl") THEN
       "AlarmHorn_Out" := 0;
   END_IF;

   IF "AlarmHorn_HOA" = 1 OR ("AlarmHorn_HOA" = 2 AND "Alarm_Horn_Ctrl") THEN
       "AlarmHorn_Out" := 1;
   END_IF;


   IF "StationInterlock_HOA" = 0 OR ("StationInterlock_HOA" = 2 AND NOT "StationInterlock_Ctrl") OR "EstopAlarm"THEN
       "StationInterlock_Out" := 0;
   END_IF;

   IF ("StationInterlock_HOA" = 1 OR ("StationInterlock_HOA" = 2 AND "StationInterlock_Ctrl"))AND NOT "EstopAlarm" THEN
       "StationInterlock_Out" := 1;
   END_IF;


   IF "Baffle_HOA" = 0 OR ("Baffle_HOA" = 2 AND NOT "Baffle_Ctrl") THEN
       "Baffle_En" := 0;
   END_IF;

   IF "Baffle_HOA" = 1 OR ("Baffle_HOA" = 2 AND "StationInterlock_Ctrl") THEN
       "Baffle_En" := 1;
   END_IF;



   //Analog outputs:
   "Scale_with_Parameters"(Input_min:=0,
                           Input_signal:="OilPump_VFD_Pct",
                           Input_max:=100,
                           Output_max:=27648,
                           Output_min:=0,
                           sv=>"OilPumpVFDsp_Out");

   "Scale_with_Parameters"(Input_min := 0,
                           Input_signal := "Baffle_Pct",
                           Input_max := 100,
                           Output_max := 27648,
                           Output_min := 0,
                           sv => "Baffle_Out");


   //Analog inputs:
   "Scale_with_Parameters"(Input_min := 0,
                           Input_signal := "OilTemp_In",
                           Input_max := 27648,
                           Output_max := 500,
                           Output_min := 0,
                           sv => "OilTemp");

   "Scale_with_Parameters"(Input_min := 0,
                           Input_signal := "OilFlow_In",
                           Input_max := 27648,
                           Output_max := 30,
                           Output_min := 0,
                           sv => "OilFlow");

   "Scale_with_Parameters"(Input_min := 0,
                           Input_signal := "RPM_In",
                           Input_max := 27648,
                           Output_max := 200,
                           Output_min := 0,
                           sv => "RPM");

   "Scale_with_Parameters"(Input_min := 0,
                           Input_signal := "Current_In",
                           Input_max := 27648,
                           Output_max := 700,
                           Output_min := 0,
                           sv => "Current");
   // Full auto Bit
   // 
   IF "Brake_HOA"=2 AND "VFD_HOA"=2 AND "Baffle_HOA"=2 AND "AlarmHorn_HOA"=2 AND "StationInterlock_HOA"=2 THEN
       "Full_Auto_Bit" := 1;
   ELSE
       "Full_Auto_Bit" := 0;
   END_IF;
END_FUNCTION_BLOCK

FUNCTION_BLOCK "IO_STL"   // FB5, STL
{ S7_Optimized_Access := 'TRUE' }
VERSION : 0.1
   VAR_TEMP
      tb1 : Bool;
      tb2 : Bool;
      tb3 : Bool;
      tb4 : Bool;
      tb5 : Bool;
   END_VAR
BEGIN

REGION Network 1
   //Digital Outputs:
         A     "OilLowFlowAlarm";
         JC    ResetPumpVFD;
         CLR;
         A     "EstopAlarm";
         JC    ResetPumpVFD;
         CLR;

         L     "VFD_HOA";
         L     0;
         ==I;
         JC    ResetPumpVFD;
         CLR;
         L     "VFD_HOA";
         L     1;
         ==I;
         JC    SetPumpVFD;
         CLR;
         L     "VFD_HOA";
         L     2;
         ==I;
         JC    AutoPumpVFD;
         CLR;


   AutoPumpVFD:A     "OilPumpVFD_Ctrl";
         JC    SetPumpVFD;
         JU    ResetPumpVFD;

   SetPumpVFD:AN    "OilLowFlowAlarm";
         AN    "EstopAlarm";
         S     "OilPumpVFDen_Out";
         JU    Brake;
   ResetPumpVFD:R     "OilPumpVFDen_Out";
         JU    Brake;

   //---------------------------------------------------------------
   Brake:L     "Brake_HOA";
         L     0;
         ==I;
         JC    ResetBrake;
         CLR;
         L     "Brake_HOA";
         L     1;
         ==I;
         JC    SetBrake;
         CLR;
         L     "Brake_HOA";
         L     2;
         ==I;
         JC    AutoBrake;
         CLR;


   AutoBrake:A     "Brake_Ctrl";
         JC    SetBrake;
         JU    ResetBrake;

   SetBrake:S     "Brake_Out";
         JU    AlarmHorn;
   ResetBrake:R     "Brake_Out";
         JU    AlarmHorn;
   //--------------------------------------------------------------
   AlarmHorn:L     "AlarmHorn_HOA";
         L     0;
         ==I;
         JC    ResetAlarm;
         CLR;
         L     "AlarmHorn_HOA";
         L     1;
         ==I;
         JC    SetAlarm;
         CLR;
         L     "AlarmHorn_HOA";
         L     2;
         ==I;
         JC    AutoAlarm;
         CLR;


   AutoAlarm:A     "Alarm_Horn_Ctrl";
         JC    SetAlarm;
         JU    ResetAlarm;

   SetAlarm:S     "AlarmHorn_Out";
         JU    Station;
   ResetAlarm:R     "AlarmHorn_Out";
         JU    Station;

   //----------------------------------------------------------------

   Station:A     "EstopAlarm";
         JC    ResetStation;
         CLR;
         L     "StationInterlock_HOA";
         L     0;
         ==I;
         JC    ResetStation;
         CLR;
         L     "StationInterlock_HOA";
         L     1;
         ==I;
         JC    SetStation;
         CLR;
         L     "StationInterlock_HOA";
         L     2;
         ==I;
         JC    AutoStation;
         CLR;


   AutoStation:A     "StationInterlock_Ctrl";
         JC    SetStation;
         JU    ResetStation;

   SetStation:AN    "EstopAlarm";
         S     "StationInterlock_Out";
         JU    Baffle;
   ResetStation:R     "StationInterlock_Out";
         JU    Baffle;

   //-----------------------------------------------------------------------
   Baffle:L     "Baffle_HOA";
         L     0;
         ==I;
         JC    ResetBaffle;
         CLR;
         L     "Baffle_HOA";
         L     1;
         ==I;
         JC    SetBaffle;
         CLR;
         L     "Baffle_HOA";
         L     2;
         ==I;
         JC    AutoBaffle;
         CLR;


   AutoBaffle:A     "Baffle_Ctrl";
         JC    SetBaffle;
         JU    ResetBaffle;

   SetBaffle:S     "Baffle_En";
         JU    AnalogOutputs;
   ResetBaffle:R     "Baffle_En";
         JU    AnalogOutputs;

   //----------------------------------------------------------------------



   //AnaloAnalog Outputs
   AnalogOutputs:CALL  "Scale_with_Parameters"
         ( Input_min    := 0,
           Input_signal := "OilPump_VFD_Pct",
           Input_max    := 100,
           Output_max   := 27648,
           Output_min   := 0,
           sv           := "OilPumpVFDsp_Out"
         );


         CALL  "Scale_with_Parameters"
         ( Input_min    := 0,
           Input_signal := "Baffle_Pct",
           Input_max    := 100,
           Output_max   := 27648,
           Output_min   := 0,
           sv           := "Baffle_Out"
         );


   //Analog inputs



   AnalogInputs:CALL  "Scale_with_Parameters"
         ( Input_min    := 0,
           Input_signal := "OilTemp_In",
           Input_max    := 27648,
           Output_max   := 500,
           Output_min   := 0,
           sv           := "OilTemp"
         );


         CALL  "Scale_with_Parameters"
         ( Input_min    := 0,
           Input_signal := "OilFlow_In",
           Input_max    := 27648,
           Output_max   := 30,
           Output_min   := 0,
           sv           := "OilFlow"
         );


         CALL  "Scale_with_Parameters"
         ( Input_min    := 0,
           Input_signal := "RPM_In",
           Input_max    := 27648,
           Output_max   := 200,
           Output_min   := 0,
           sv           := "RPM"
         );


         CALL  "Scale_with_Parameters"
         ( Input_min    := 0,
           Input_signal := "Current_In",
           Input_max    := 27648,
           Output_max   := 700,
           Output_min   := 0,
           sv           := "Current"
         );

   //---------------Full Auto Bit---------------------------------
         L     "Baffle_HOA";
         L     2;
         ==I;
         NOT;
         JC    ResetFullAuto;
         CLR;
         L     "Brake_HOA";
         L     2;
         ==I;
         NOT;
         JC    ResetFullAuto;
         CLR;
         L     "StationInterlock_HOA";
         L     2;
         ==I;
         NOT;
         JC    ResetFullAuto;
         CLR;
         L     "VFD_HOA";
         L     2;
         ==I;
         NOT;
         JC    ResetFullAuto;
         CLR;
         L     "AlarmHorn_HOA";
         L     2;
         ==I;
         NOT;
         JC    ResetFullAuto;
         JU    SetFullAuto;
   SetFullAuto:SET;
         S     "Full_Auto_Bit";
         BE;
   ResetFullAuto:SET;
         R     "Full_Auto_Bit";
         BE;
END_REGION
END_FUNCTION_BLOCK

FUNCTION_BLOCK "ALARMS_LAD"   // FB6, LAD
{ S7_Optimized_Access := 'TRUE' }
VERSION : 0.1
   VAR RETAIN
      ONS4 : Bool;
      ONS5 : Bool;
      ONS7 : Bool;
      ONS6 : Bool;
      ONS8 : Bool;
      ONS9 : Bool;
   END_VAR
   VAR
      ONS10 : Bool;
      OS1 : Bool;
      AlarmHornTrigger : Bool;
   END_VAR
   VAR_TEMP
      OFD : Int;
      OilFlow_AT : Bool;
      tv1 : Time;
      OCD : Int;
      tv2 : Time;
      Overcurent_AT : Bool;
      HOTD : Int;
      tv3 : Time;
      HighOilTemp_AT : Bool;
      ROD : Int;
      tv4 : Time;
      RotorOverspeed_AT : Bool;
      HOFD : Int;
      tv5 : Time;
      OilFlowHigh_AT : Bool;
      BFD : Int;
      tv6 : Time;
      BF_AT : Bool;
      Estop_AT : Bool;
   END_VAR
   VAR_TEMP   // added for the SCL form of the ladder/FBD networks
      _w1 : Bool;
      _w2 : Bool;
   END_VAR
BEGIN

REGION Network 1
   // Low Oil Flow Alarm
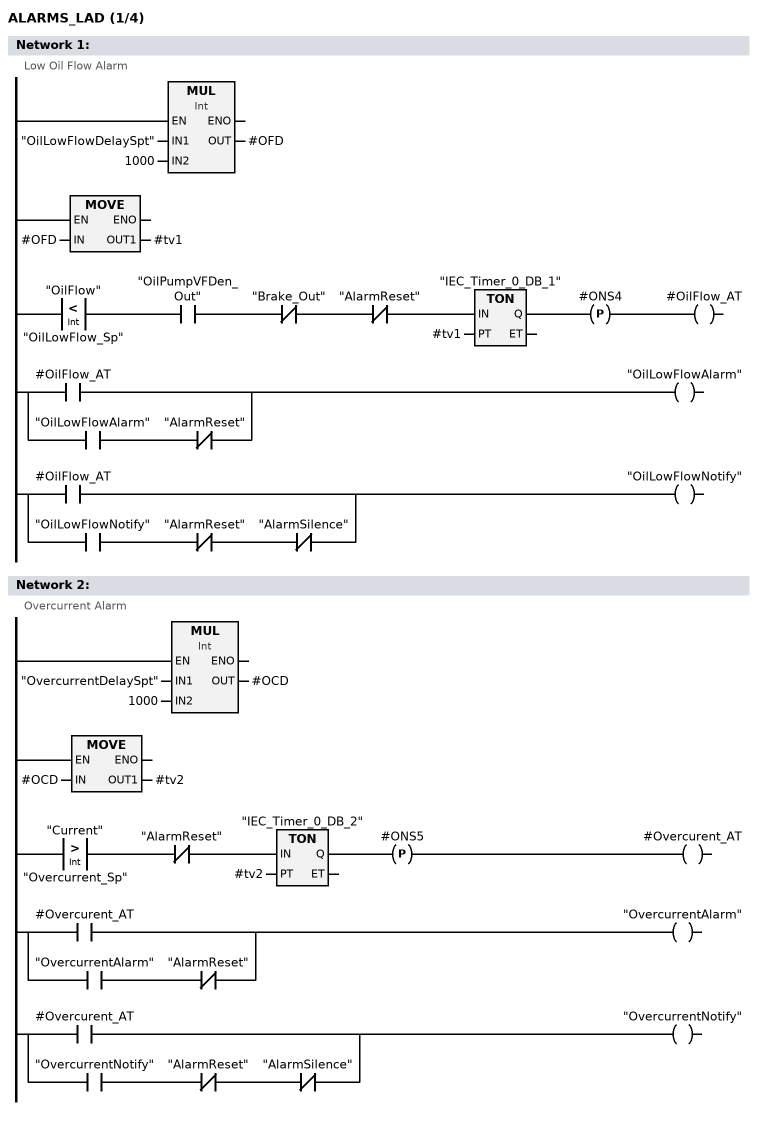
   #OFD := "OilLowFlowDelaySpt" * 1000;
   #tv1 := #OFD;
   "IEC_Timer_0_DB_1".TON(IN := ("OilFlow" < "OilLowFlow_Sp") AND "OilPumpVFDen_Out" AND NOT "Brake_Out" AND NOT "AlarmReset",
                          PT := #tv1);
   #_w1 := "IEC_Timer_0_DB_1".Q AND NOT #ONS4;   // rising edge
   #ONS4 := "IEC_Timer_0_DB_1".Q;
   #OilFlow_AT := #_w1;
   "OilLowFlowAlarm" := #OilFlow_AT OR ("OilLowFlowAlarm" AND NOT "AlarmReset");
   "OilLowFlowNotify" := #OilFlow_AT OR ("OilLowFlowNotify" AND NOT "AlarmReset" AND NOT "AlarmSilence");
END_REGION

REGION Network 2
   // Overcurrent Alarm
   #OCD := "OvercurrentDelaySpt" * 1000;
   #tv2 := #OCD;
   "IEC_Timer_0_DB_2".TON(IN := ("Current" > "Overcurrent_Sp") AND NOT "AlarmReset", PT := #tv2);
   #_w1 := "IEC_Timer_0_DB_2".Q AND NOT #ONS5;   // rising edge
   #ONS5 := "IEC_Timer_0_DB_2".Q;
   #Overcurent_AT := #_w1;
   "OvercurrentAlarm" := #Overcurent_AT OR ("OvercurrentAlarm" AND NOT "AlarmReset");
   "OvercurrentNotify" := #Overcurent_AT OR ("OvercurrentNotify" AND NOT "AlarmReset" AND NOT "AlarmSilence");
END_REGION

REGION Network 3
   // High Oil Temp.
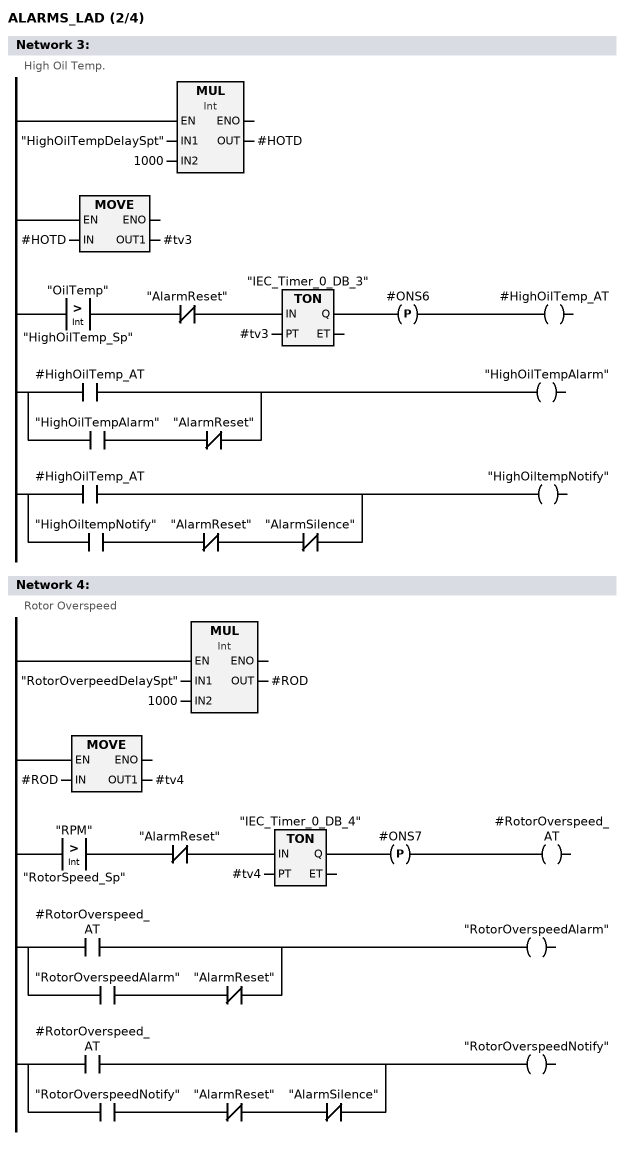
   #HOTD := "HighOilTempDelaySpt" * 1000;
   #tv3 := #HOTD;
   "IEC_Timer_0_DB_3".TON(IN := ("OilTemp" > "HighOilTemp_Sp") AND NOT "AlarmReset", PT := #tv3);
   #_w1 := "IEC_Timer_0_DB_3".Q AND NOT #ONS6;   // rising edge
   #ONS6 := "IEC_Timer_0_DB_3".Q;
   #HighOilTemp_AT := #_w1;
   "HighOilTempAlarm" := #HighOilTemp_AT OR ("HighOilTempAlarm" AND NOT "AlarmReset");
   "HighOiltempNotify" := #HighOilTemp_AT OR ("HighOiltempNotify" AND NOT "AlarmReset" AND NOT "AlarmSilence");
END_REGION

REGION Network 4
   // Rotor Overspeed
   #ROD := "RotorOverpeedDelaySpt" * 1000;
   #tv4 := #ROD;
   "IEC_Timer_0_DB_4".TON(IN := ("RPM" > "RotorSpeed_Sp") AND NOT "AlarmReset", PT := #tv4);
   #_w1 := "IEC_Timer_0_DB_4".Q AND NOT #ONS7;   // rising edge
   #ONS7 := "IEC_Timer_0_DB_4".Q;
   #RotorOverspeed_AT := #_w1;
   "RotorOverspeedAlarm" := #RotorOverspeed_AT OR ("RotorOverspeedAlarm" AND NOT "AlarmReset");
   "RotorOverspeedNotify" := #RotorOverspeed_AT OR ("RotorOverspeedNotify" AND NOT "AlarmReset" AND NOT "AlarmSilence");
END_REGION

REGION Network 5
   // High Oil Flow Alarm
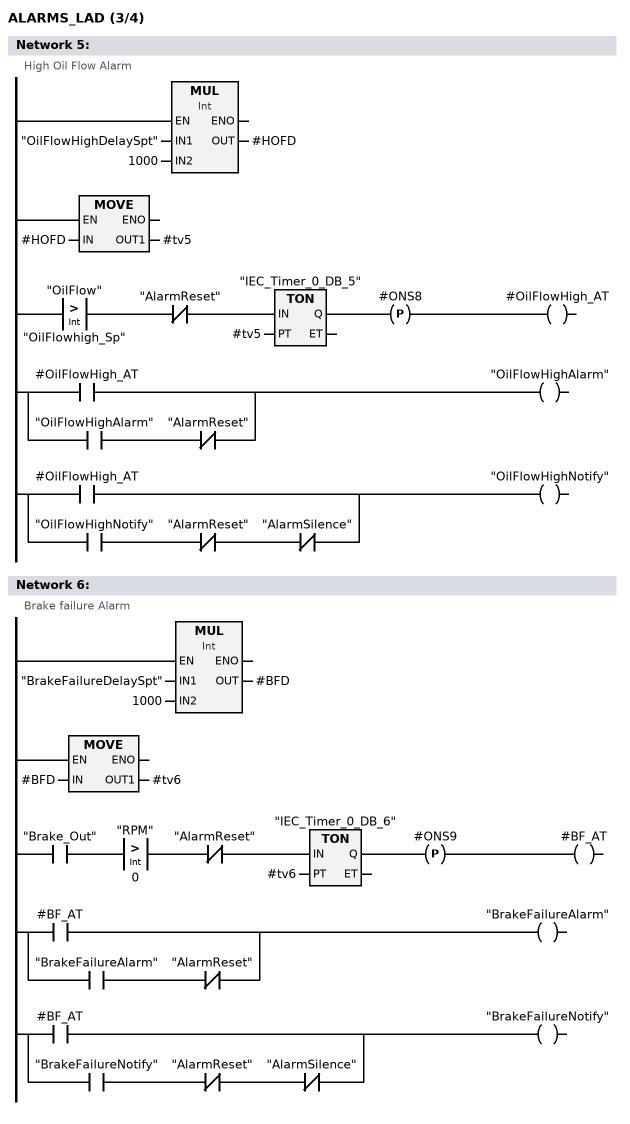
   #HOFD := "OilFlowHighDelaySpt" * 1000;
   #tv5 := #HOFD;
   "IEC_Timer_0_DB_5".TON(IN := ("OilFlow" > "OilFlowhigh_Sp") AND NOT "AlarmReset", PT := #tv5);
   #_w1 := "IEC_Timer_0_DB_5".Q AND NOT #ONS8;   // rising edge
   #ONS8 := "IEC_Timer_0_DB_5".Q;
   #OilFlowHigh_AT := #_w1;
   "OilFlowHighAlarm" := #OilFlowHigh_AT OR ("OilFlowHighAlarm" AND NOT "AlarmReset");
   "OilFlowHighNotify" := #OilFlowHigh_AT OR ("OilFlowHighNotify" AND NOT "AlarmReset" AND NOT "AlarmSilence");
END_REGION

REGION Network 6
   // Brake failure Alarm
   #BFD := "BrakeFailureDelaySpt" * 1000;
   #tv6 := #BFD;
   "IEC_Timer_0_DB_6".TON(IN := "Brake_Out" AND ("RPM" > 0) AND NOT "AlarmReset", PT := #tv6);
   #_w1 := "IEC_Timer_0_DB_6".Q AND NOT #ONS9;   // rising edge
   #ONS9 := "IEC_Timer_0_DB_6".Q;
   #BF_AT := #_w1;
   "BrakeFailureAlarm" := #BF_AT OR ("BrakeFailureAlarm" AND NOT "AlarmReset");
   "BrakeFailureNotify" := #BF_AT OR ("BrakeFailureNotify" AND NOT "AlarmReset" AND NOT "AlarmSilence");
END_REGION

REGION Network 7
   // Estop
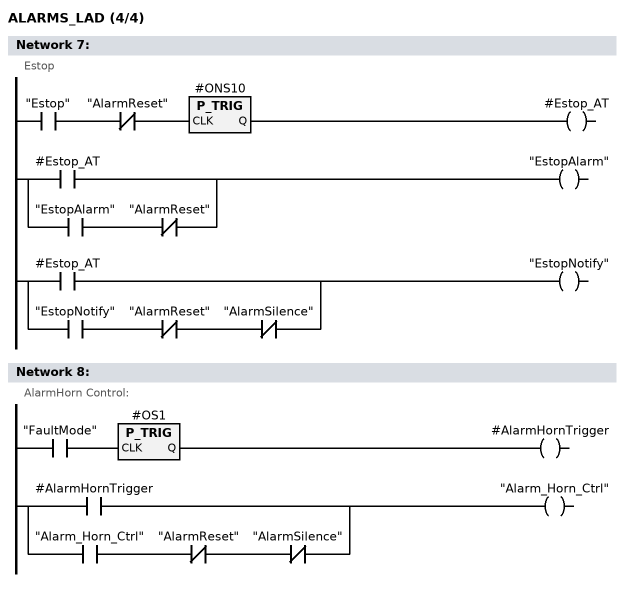
   RUNG wire#powerrail
      Contact( "Estop" )
      I_Contact( "AlarmReset" )
      P_Trig( #ONS10 )
      Coil( #Estop_AT )
   END_RUNG
   RUNG wire#powerrail
      Contact( #Estop_AT )
      wire#w1
      Coil( "EstopAlarm" )
   END_RUNG
   RUNG wire#powerrail
      Contact( "EstopAlarm" )
      I_Contact( "AlarmReset" )
   END_RUNG wire#w1
   RUNG wire#powerrail
      Contact( #Estop_AT )
      wire#w2
      Coil( "EstopNotify" )
   END_RUNG
   RUNG wire#powerrail
      Contact( "EstopNotify" )
      I_Contact( "AlarmReset" )
      I_Contact( "AlarmSilence" )
   END_RUNG wire#w2
   // the same network as SCL:
   #_w1 := "Estop" AND NOT "AlarmReset";
   #_w2 := #_w1 AND NOT #ONS10;   // rising edge
   #ONS10 := #_w1;
   #Estop_AT := #_w2;
   "EstopAlarm" := #Estop_AT OR ("EstopAlarm" AND NOT "AlarmReset");
   "EstopNotify" := #Estop_AT OR ("EstopNotify" AND NOT "AlarmReset" AND NOT "AlarmSilence");
END_REGION

REGION Network 8
   // AlarmHorn Control:
   RUNG wire#powerrail
      Contact( "FaultMode" )
      P_Trig( #OS1 )
      Coil( #AlarmHornTrigger )
   END_RUNG
   RUNG wire#powerrail
      Contact( #AlarmHornTrigger )
      wire#w1
      Coil( "Alarm_Horn_Ctrl" )
   END_RUNG
   RUNG wire#powerrail
      Contact( "Alarm_Horn_Ctrl" )
      I_Contact( "AlarmReset" )
      I_Contact( "AlarmSilence" )
   END_RUNG wire#w1
   // the same network as SCL:
   #_w1 := "FaultMode" AND NOT #OS1;   // rising edge
   #OS1 := "FaultMode";
   #AlarmHornTrigger := #_w1;
   "Alarm_Horn_Ctrl" := #AlarmHornTrigger OR ("Alarm_Horn_Ctrl" AND NOT "AlarmReset" AND NOT "AlarmSilence");
END_REGION
END_FUNCTION_BLOCK

FUNCTION_BLOCK "ALARMS_FBD"   // FB7, FBD
{ S7_Optimized_Access := 'TRUE' }
VERSION : 0.1
   VAR
      ONS4 : Bool;
      ONS5 : Bool;
      ONS6 : Bool;
      ONS7 : Bool;
      ONS8 : Bool;
      ONS9 : Bool;
      ONS10 : Bool;
      ONS11 : Bool;
      OS1 : Bool;
      AlarmHornTrigger : Bool;
   END_VAR
   VAR_TEMP
      tv1 : Int;
      OFLD : Time;
      tv2 : Int;
      OCD : Time;
      tv3 : Int;
      HOTD : Time;
      tv4 : Int;
      ROD : Time;
      tv5 : Int;
      HOFD : Time;
      tv6 : Int;
      BFD : Time;
   END_VAR
   VAR_TEMP   // added for the SCL form of the ladder/FBD networks
      _w1 : Bool;
      _w2 : Bool;
   END_VAR
BEGIN

REGION Network 1
   // Low Oil Flow
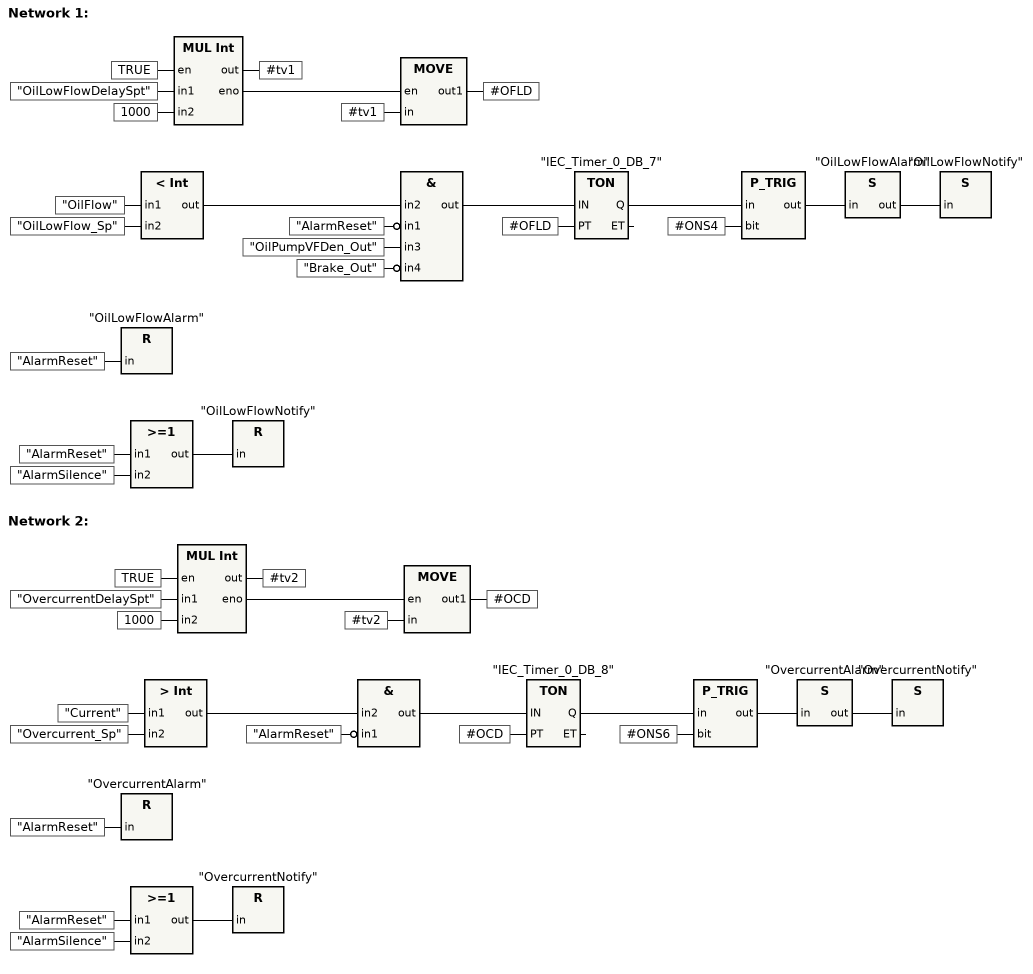
   IF TRUE THEN
       #tv1 := "OilLowFlowDelaySpt" * 1000;
       #OFLD := #tv1;
   END_IF;
   "IEC_Timer_0_DB_7".TON(IN := ("OilFlow" < "OilLowFlow_Sp") AND NOT "AlarmReset" AND "OilPumpVFDen_Out" AND NOT "Brake_Out",
                          PT := #OFLD);
   #_w1 := "IEC_Timer_0_DB_7".Q AND NOT #ONS4;   // rising edge
   #ONS4 := "IEC_Timer_0_DB_7".Q;
   IF #_w1 THEN
       "OilLowFlowAlarm" := TRUE;
       "OilLowFlowNotify" := TRUE;
   END_IF;
   IF "AlarmReset" THEN "OilLowFlowAlarm" := FALSE; END_IF;
   IF "AlarmReset" OR "AlarmSilence" THEN "OilLowFlowNotify" := FALSE; END_IF;
END_REGION

REGION Network 2
   // Overcurrent Alarm:
   IF TRUE THEN
       #tv2 := "OvercurrentDelaySpt" * 1000;
       #OCD := #tv2;
   END_IF;
   "IEC_Timer_0_DB_8".TON(IN := ("Current" > "Overcurrent_Sp") AND NOT "AlarmReset", PT := #OCD);
   #_w1 := "IEC_Timer_0_DB_8".Q AND NOT #ONS6;   // rising edge
   #ONS6 := "IEC_Timer_0_DB_8".Q;
   IF #_w1 THEN
       "OvercurrentAlarm" := TRUE;
       "OvercurrentNotify" := TRUE;
   END_IF;
   IF "AlarmReset" THEN "OvercurrentAlarm" := FALSE; END_IF;
   IF "AlarmReset" OR "AlarmSilence" THEN "OvercurrentNotify" := FALSE; END_IF;
END_REGION

REGION Network 3
   // HighOiltemp Alarm:
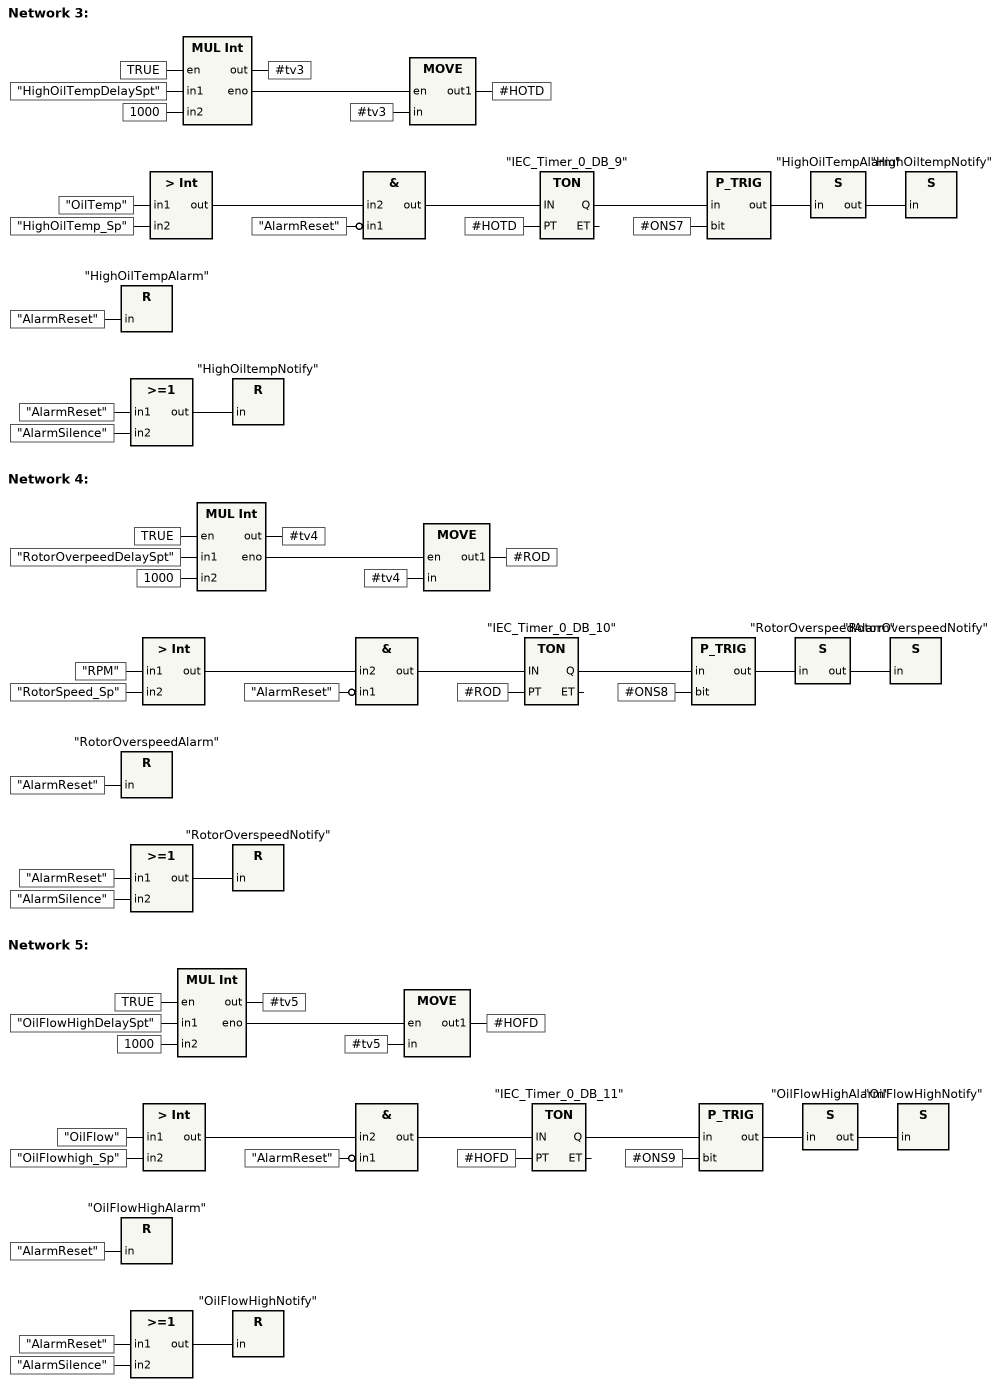
   IF TRUE THEN
       #tv3 := "HighOilTempDelaySpt" * 1000;
       #HOTD := #tv3;
   END_IF;
   "IEC_Timer_0_DB_9".TON(IN := ("OilTemp" > "HighOilTemp_Sp") AND NOT "AlarmReset", PT := #HOTD);
   #_w1 := "IEC_Timer_0_DB_9".Q AND NOT #ONS7;   // rising edge
   #ONS7 := "IEC_Timer_0_DB_9".Q;
   IF #_w1 THEN
       "HighOilTempAlarm" := TRUE;
       "HighOiltempNotify" := TRUE;
   END_IF;
   IF "AlarmReset" THEN "HighOilTempAlarm" := FALSE; END_IF;
   IF "AlarmReset" OR "AlarmSilence" THEN "HighOiltempNotify" := FALSE; END_IF;
END_REGION

REGION Network 4
   // Rotor Overspeed:
   IF TRUE THEN
       #tv4 := "RotorOverpeedDelaySpt" * 1000;
       #ROD := #tv4;
   END_IF;
   "IEC_Timer_0_DB_10".TON(IN := ("RPM" > "RotorSpeed_Sp") AND NOT "AlarmReset", PT := #ROD);
   #_w1 := "IEC_Timer_0_DB_10".Q AND NOT #ONS8;   // rising edge
   #ONS8 := "IEC_Timer_0_DB_10".Q;
   IF #_w1 THEN
       "RotorOverspeedAlarm" := TRUE;
       "RotorOverspeedNotify" := TRUE;
   END_IF;
   IF "AlarmReset" THEN "RotorOverspeedAlarm" := FALSE; END_IF;
   IF "AlarmReset" OR "AlarmSilence" THEN "RotorOverspeedNotify" := FALSE; END_IF;
END_REGION

REGION Network 5
   // High Oil Flow Alarm
   IF TRUE THEN
       #tv5 := "OilFlowHighDelaySpt" * 1000;
       #HOFD := #tv5;
   END_IF;
   "IEC_Timer_0_DB_11".TON(IN := ("OilFlow" > "OilFlowhigh_Sp") AND NOT "AlarmReset", PT := #HOFD);
   #_w1 := "IEC_Timer_0_DB_11".Q AND NOT #ONS9;   // rising edge
   #ONS9 := "IEC_Timer_0_DB_11".Q;
   IF #_w1 THEN
       "OilFlowHighAlarm" := TRUE;
       "OilFlowHighNotify" := TRUE;
   END_IF;
   IF "AlarmReset" THEN "OilFlowHighAlarm" := FALSE; END_IF;
   IF "AlarmReset" OR "AlarmSilence" THEN "OilFlowHighNotify" := FALSE; END_IF;
END_REGION

REGION Network 6
   // Brake failure Alarm:
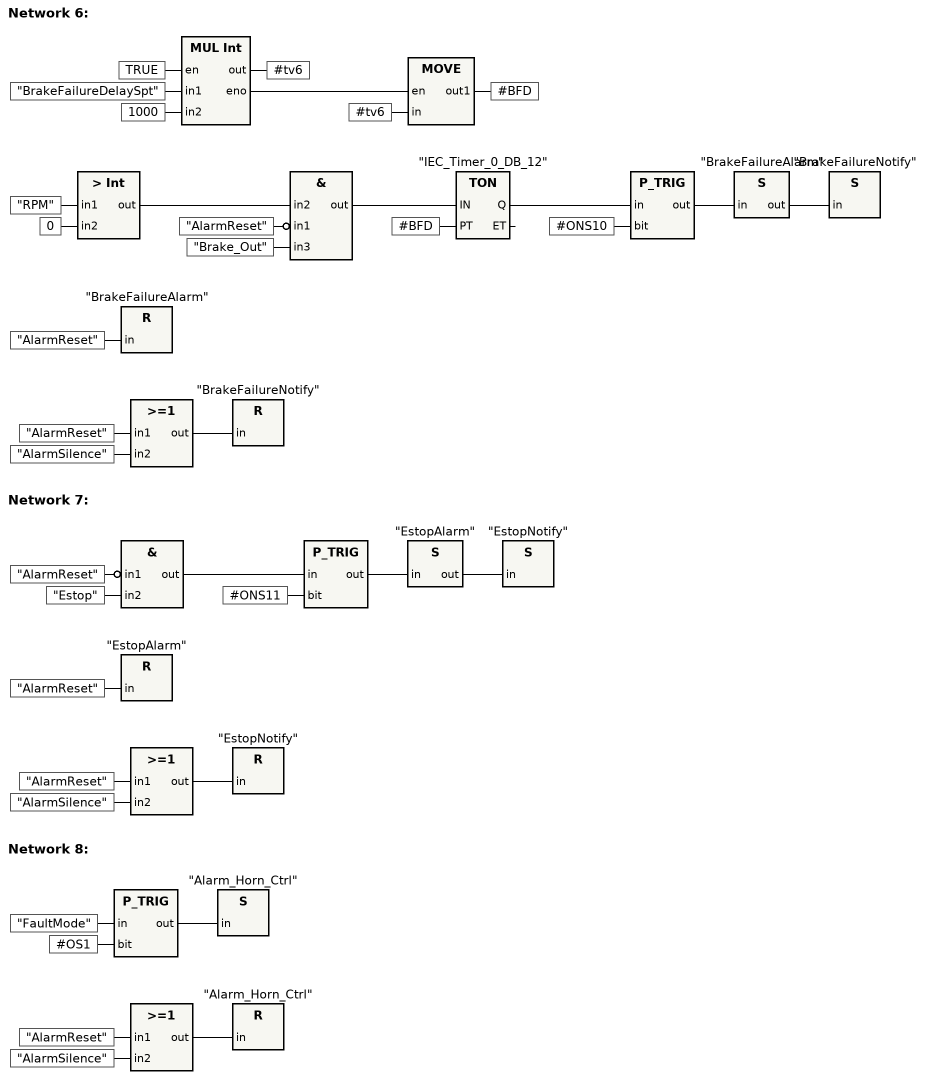
   IF TRUE THEN
       #tv6 := "BrakeFailureDelaySpt" * 1000;
       #BFD := #tv6;
   END_IF;
   "IEC_Timer_0_DB_12".TON(IN := ("RPM" > 0) AND NOT "AlarmReset" AND "Brake_Out", PT := #BFD);
   #_w1 := "IEC_Timer_0_DB_12".Q AND NOT #ONS10;   // rising edge
   #ONS10 := "IEC_Timer_0_DB_12".Q;
   IF #_w1 THEN
       "BrakeFailureAlarm" := TRUE;
       "BrakeFailureNotify" := TRUE;
   END_IF;
   IF "AlarmReset" THEN "BrakeFailureAlarm" := FALSE; END_IF;
   IF "AlarmReset" OR "AlarmSilence" THEN "BrakeFailureNotify" := FALSE; END_IF;
END_REGION

REGION Network 7
   // Estop:
   #_w1 := NOT "AlarmReset" AND "Estop";
   #_w2 := #_w1 AND NOT #ONS11;   // rising edge
   #ONS11 := #_w1;
   IF #_w2 THEN
       "EstopAlarm" := TRUE;
       "EstopNotify" := TRUE;
   END_IF;
   IF "AlarmReset" THEN "EstopAlarm" := FALSE; END_IF;
   IF "AlarmReset" OR "AlarmSilence" THEN "EstopNotify" := FALSE; END_IF;
END_REGION

REGION Network 8
   // AlarmHorn Control:
   #_w1 := "FaultMode" AND NOT #OS1;   // rising edge
   #OS1 := "FaultMode";
   IF #_w1 THEN "Alarm_Horn_Ctrl" := TRUE; END_IF;
   IF "AlarmReset" OR "AlarmSilence" THEN "Alarm_Horn_Ctrl" := FALSE; END_IF;
END_REGION
END_FUNCTION_BLOCK

FUNCTION_BLOCK "ALARMS_SCL"   // FB8, SCL
{ S7_Optimized_Access := 'TRUE' }
VERSION : 0.1
   VAR_TEMP
      t1 : Time;
      t2 : Time;
      t3 : Time;
      t4 : Time;
      t5 : Time;
      t6 : Time;
      t7 : Time;
      et1 : Time;
      et2 : Time;
      et3 : Time;
      et4 : Time;
      et5 : Time;
      et6 : Time;
      et7 : Time;
      OLFT : Bool;
      OCT : Bool;
      HOTT : Bool;
      ROT : Bool;
      HOFT : Bool;
      BFT : Bool;
   END_VAR
BEGIN
   //Oil low flow Alarm

   IF "OilPumpVFDen_Out" AND "OilFlow"< "OilLowFlow_Sp" AND NOT"AlarmReset" AND NOT "Brake_Out" AND NOT "OilLowFlowAlarm"  THEN

      "time conversion"(timein:= "OilLowFlowDelaySpt",
                        time_out=>#t1);


   "IEC_Timer_0_DB_13".TON(IN:=TRUE,
                             PT:=#t1,
                             Q=>#OLFT,
                             ET=>#et1);
   ELSE
      RESET_TIMER("IEC_Timer_0_DB_13");


   END_IF;
   IF #OLFT  THEN
       "OilLowFlowAlarm" := 1;
       "OilLowFlowNotify" := 1;
   END_IF;
   IF "OilLowFlowAlarm" AND "AlarmReset" THEN
       "OilLowFlowAlarm" := 0;
       "OilLowFlowNotify" := 0;
   END_IF;
   IF "OilLowFlowNotify" AND "AlarmSilence" THEN
       "OilLowFlowNotify" := 0;
   END_IF;

   //Overcurrent alarm:

   IF "Current" > "Overcurrent_Sp" AND NOT "OvercurrentAlarm" AND NOT "AlarmReset" THEN

       "time conversion"(timein := "OvercurrentDelaySpt",
                         time_out => #t2);
      "IEC_Timer_0_DB_15".TON(IN:=TRUE,
                              PT:=#t2,
                              Q=>#OCT,
                              ET=>#et2);
   ELSE
       RESET_TIMER("IEC_Timer_0_DB_15");

   END_IF;
   IF #OCT THEN
       "OvercurrentAlarm" := 1;
       "OvercurrentNotify" := 1;
   END_IF;
   IF "OvercurrentAlarm" AND "AlarmReset" THEN
       "OvercurrentAlarm" := 0;
       "OvercurrentNotify" := 0;
   END_IF;
   IF "OvercurrentNotify" AND "AlarmSilence" THEN
       "OvercurrentNotify" := 0;
   END_IF;

   //High Oil Temp Alarm:


   IF "OilTemp" > "HighOilTemp_Sp" AND NOT "HighOilTempAlarm" AND NOT "AlarmReset" THEN

       "time conversion"(timein := "HighOilTempDelaySpt",
                         time_out => #t3);
     "IEC_Timer_0_DB_16".TON(IN:=TRUE,
                             PT:=#t3,
                             Q=>#HOTT,
                             ET=>#et3);

   ELSE
       RESET_TIMER("IEC_Timer_0_DB_16");

   END_IF;
   IF #HOTT THEN
       "HighOilTempAlarm" := 1;
       "HighOiltempNotify" := 1;
   END_IF;
   IF "HighOilTempAlarm" AND "AlarmReset" THEN
       "HighOilTempAlarm" := 0;
       "HighOiltempNotify" := 0;
   END_IF;
   IF "HighOiltempNotify" AND "AlarmSilence" THEN
       "HighOiltempNotify" := 0;
   END_IF;

   //Rotor overspeed Alarm:

   IF "RPM" > "RotorSpeed_Sp" AND NOT "RotorOverspeedAlarm" AND NOT"AlarmReset" THEN

       "time conversion"(timein := "RotorOverpeedDelaySpt",
                         time_out => #t4);
    "IEC_Timer_0_DB_17".TON(IN:=TRUE,
                            PT:=#t4,
                            Q=>#ROT,
                            ET=>#et4);
   ELSE
       RESET_TIMER("IEC_Timer_0_DB_17");


   END_IF;
   IF #ROT THEN
       "RotorOverspeedAlarm" := 1;
       "RotorOverspeedNotify" := 1;
   END_IF;
   IF "RotorOverspeedAlarm" AND "AlarmReset" THEN
       "RotorOverspeedAlarm" := 0;
       "RotorOverspeedNotify" := 0;
   END_IF;
   IF "RotorOverspeedNotify" AND "AlarmSilence" THEN
       "RotorOverspeedNotify" := 0;
   END_IF;

   //Oil High Flow Alarm:

   IF "OilFlow" > "OilFlowhigh_Sp" AND NOT "OilFlowHighAlarm" AND NOT "AlarmReset" THEN

       "time conversion"(timein := "OilFlowHighDelaySpt",
                         time_out => #t5);
     "IEC_Timer_0_DB_19".TON(IN:=TRUE,
                             PT:=#t5,
                             Q=>#HOFT,
                             ET=>#et5);
   ELSE
       RESET_TIMER("IEC_Timer_0_DB_19");



   END_IF;
   IF #HOFT THEN
       "OilFlowHighAlarm" := 1;
       "OilFlowHighNotify" := 1;
   END_IF;
   IF "OilFlowHighAlarm" AND "AlarmReset" THEN
       "OilFlowHighAlarm" := 0;
       "OilFlowHighNotify" := 0;
   END_IF;
   IF "OilFlowHighNotify" AND "AlarmSilence" THEN
       "OilFlowHighNotify" := 0;
   END_IF;

   //Brake Failure Alarm:


   IF "RPM" > 0 AND "Brake_Out"AND NOT "BrakeFailureAlarm" AND NOT"AlarmReset" THEN

       "time conversion"(timein := "BrakeFailureDelaySpt",
                         time_out => #t6);
     "IEC_Timer_0_DB_20".TON(IN:=TRUE,
                             PT:=#t6,
                             Q=>#BFT,
                             ET=>#et6);
   ELSE
       RESET_TIMER("IEC_Timer_0_DB_20");


   END_IF;
   IF #BFT THEN
       "BrakeFailureAlarm" := 1;
       "BrakeFailureNotify" := 1;
   END_IF;
   IF "BrakeFailureAlarm" AND "AlarmReset" THEN
       "BrakeFailureAlarm" := 0;
       "BrakeFailureNotify" := 0;
   END_IF;
   IF "BrakeFailureNotify" AND "AlarmSilence" THEN
       "BrakeFailureNotify" := 0;
   END_IF;

   //Estop alarm:

   IF "Estop"  AND NOT "EstopAlarm" AND NOT"AlarmReset" THEN
       "EstopAlarm" := 1;
       "EstopNotify" := 1;
   END_IF;
   IF "EstopAlarm" AND "AlarmReset" THEN
       "EstopAlarm" := 0;
       "EstopNotify" := 0;
   END_IF;
   IF "EstopNotify" AND "AlarmSilence" THEN
       "EstopNotify" := 0;
   END_IF;


   //Alarm Horn Control

   IF "FaultMode" AND NOT "Alarm_Horn_Ctrl"THEN
       "Alarm_Horn_Ctrl" := 1;

   END_IF;
   IF "Alarm_Horn_Ctrl" AND ("AlarmReset" OR "AlarmSilence") THEN
       "Alarm_Horn_Ctrl" := 0;
   END_IF;
END_FUNCTION_BLOCK

FUNCTION_BLOCK "ALARMS_STL"   // FB9, STL
{ S7_Optimized_Access := 'TRUE' }
VERSION : 0.1
   VAR
      ONS4 : Bool;
      ONS5 : Bool;
      ONS6 : Bool;
      ONS7 : Bool;
      ONS8 : Bool;
      ONS9 : Bool;
      ONS10 : Bool;
      ONS11 : Bool;
      ONS12 : Bool;
      ONS13 : Bool;
      ONS14 : Bool;
      ONS15 : Bool;
      ONS16 : Bool;
      ONS17 : Bool;
      ONS18 : Bool;
      OS1 : Bool;
      OS2 : Bool;
      OS3 : Bool;
   END_VAR
   VAR_TEMP
      t1 : Time;
      t2 : Time;
      t3 : Time;
      t4 : Time;
      t5 : Time;
      t6 : Time;
      t7 : Time;
      et1 : Time;
      et2 : Time;
      et3 : Time;
      et4 : Time;
      et5 : Time;
      et6 : Time;
      et7 : Time;
      OLFT : Bool;
      OCT : Bool;
      HOTT : Bool;
      ROT : Bool;
      HOFT : Bool;
      BFT : Bool;
   END_VAR
BEGIN

REGION Network 1
   // Oil LowFlow Alarm:
         L     "OilFlow";
         L     "OilLowFlow_Sp";
         <I;
         A     "OilPumpVFDen_Out";
         AN    "Brake_Out";
         AN    "AlarmReset";
         AN    "OilLowFlowAlarm";
         JC    OLFTimer;
         CALL  RESET_TIMER
         ( "TIMER" := "IEC_Timer_0_DB_21"
         );

         CLR;
         A     "OilLowFlowAlarm";
         A     "AlarmReset";
         FP    #ONS4;
         JC    ResetOLFAlarm;
         CLR;
         A     "OilLowFlowNotify";
         A     "AlarmSilence";
         FP    #ONS5;
         JC    ResetOLFNotify;
         JU    OvercurrentAlarm;

   OLFTimer:CALL  "time conversion"
         ( timein   := "OilLowFlowDelaySpt",
           time_out := #t1
         );

         CALL  TON, "IEC_Timer_0_DB_21"
         ( IN := TRUE,
           PT := #t1,
           Q  := #OLFT,
           ET := #et1
         );
         A     #OLFT;
         JC    SetOLFAlarm;
         JU    OvercurrentAlarm;
   SetOLFAlarm:SET;
         S     "OilLowFlowAlarm";
         S     "OilLowFlowNotify";
         JU    OvercurrentAlarm;
   ResetOLFAlarm:R     "OilLowFlowAlarm";
         R     "OilLowFlowNotify";
         JU    OvercurrentAlarm;
   ResetOLFNotify:R     "OilLowFlowNotify";
         JU    OvercurrentAlarm;

   //-------------------------------------------------
   OvercurrentAlarm:L     "Current";
         L     "Overcurrent_Sp";
         >I;
         AN    "AlarmReset";
         AN    "OvercurrentAlarm";
         JC    OCTimer;
         CALL  RESET_TIMER
         ( "TIMER" := "IEC_Timer_0_DB_22"
         );

         CLR;
         A     "OvercurrentAlarm";
         A     "AlarmReset";
         FP    #ONS6;
         JC    ResetOCAlarm;
         CLR;
         A     "OvercurrentNotify";
         A     "AlarmSilence";
         FP    #ONS7;
         JC    ResetOCNotify;
         JU    HighOilTempAlarm;

   OCTimer:CALL  "time conversion"
         ( timein   := "OvercurrentDelaySpt",
           time_out := #t2
         );


         CALL  TON, "IEC_Timer_0_DB_22"
         ( IN := TRUE,
           PT := #t2,
           Q  := #OCT,
           ET := #et2
         );
         A     #OCT;
         JC    SetOCAlarm;
         JU    HighOilTempAlarm;
   SetOCAlarm:SET;
         S     "OvercurrentAlarm";
         S     "OvercurrentNotify";
         JU    HighOilTempAlarm;
   ResetOCAlarm:R     "OvercurrentAlarm";
         R     "OvercurrentNotify";
         JU    HighOilTempAlarm;
   ResetOCNotify:R     "OvercurrentNotify";
         JU    HighOilTempAlarm;
   //---------------------------------------------------------------
   HighOilTempAlarm:L     "OilTemp";
         L     "HighOilTemp_Sp";
         >I;
         AN    "AlarmReset";
         AN    "HighOilTempAlarm";
         JC    HOTTimer;
         CALL  RESET_TIMER
         ( "TIMER" := "IEC_Timer_0_DB_23"
         );

         CLR;
         A     "HighOilTempAlarm";
         A     "AlarmReset";
         FP    #ONS8;
         JC    ResetHOTAlarm;
         CLR;
         A     "HighOiltempNotify";
         A     "AlarmSilence";
         FP    #ONS9;
         JC    ResetHOTNotify;
         JU    RotorOverspeedAlarm;

   HOTTimer:CALL  "time conversion"
         ( timein   := "HighOilTempDelaySpt",
           time_out := #t3
         );



         CALL  TON, "IEC_Timer_0_DB_23"
         ( IN := TRUE,
           PT := #t3,
           Q  := #HOTT,
           ET := #et3
         );
         A     #HOTT;
         JC    SetHOTAlarm;
         JU    RotorOverspeedAlarm;
   SetHOTAlarm:SET;
         S     "HighOilTempAlarm";
         S     "HighOiltempNotify";
         JU    RotorOverspeedAlarm;
   ResetHOTAlarm:R     "HighOilTempAlarm";
         R     "HighOiltempNotify";
         JU    RotorOverspeedAlarm;
   ResetHOTNotify:R     "HighOiltempNotify";
         JU    RotorOverspeedAlarm;
   //--------------------------------------------------------------

   RotorOverspeedAlarm:L     "RPM";
         L     "RotorSpeed_Sp";
         >I;
         AN    "AlarmReset";
         AN    "RotorOverspeedAlarm";
         JC    ROTimer;
         CALL  RESET_TIMER
         ( "TIMER" := "IEC_Timer_0_DB_24"
         );
         CLR;
         A     "RotorOverspeedAlarm";
         A     "AlarmReset";
         FP    #ONS10;
         JC    ResetROAlarm;
         CLR;
         A     "RotorOverspeedNotify";
         A     "AlarmSilence";
         FP    #ONS11;
         JC    ResetRONotify;
         CLR;
         JU    HighOilFlowAlarm;

   ROTimer:CALL  "time conversion"
         ( timein   := "RotorOverpeedDelaySpt",
           time_out := #t4
         );
         CALL  TON, "IEC_Timer_0_DB_24"
         ( IN := TRUE,
           PT := #t4,
           Q  := #ROT,
           ET := #et4
         );


         A     #ROT;
         JC    SetROAlarm;
         JU    HighOilFlowAlarm;
   SetROAlarm:SET;
         S     "RotorOverspeedAlarm";
         S     "RotorOverspeedNotify";
         JU    HighOilFlowAlarm;
   ResetROAlarm:R     "RotorOverspeedAlarm";
         R     "RotorOverspeedNotify";
         JU    HighOilFlowAlarm;
   ResetRONotify:R     "RotorOverspeedNotify";
         JU    HighOilFlowAlarm;
   //--------------------------------------------------------------------------
   HighOilFlowAlarm:L     "OilFlow";
         L     "OilFlowhigh_Sp";
         >I;
         AN    "AlarmReset";
         AN    "OilFlowHighAlarm";
         JC    HOFTimer;
         CALL  RESET_TIMER
         ( "TIMER" := "IEC_Timer_0_DB_26"
         );

         CLR;
         A     "OilFlowHighAlarm";
         A     "AlarmReset";
         FP    #ONS12;
         JC    ResetHOFAlarm;
         CLR;
         A     "OilFlowHighNotify";
         A     "AlarmSilence";
         FP    #ONS13;
         JC    ResetHOFNotify;
         JU    BrakefailureAlarm;

   HOFTimer:CALL  "time conversion"
         ( timein   := "HighOilTempDelaySpt",
           time_out := #t5
         );

         CALL  TON, "IEC_Timer_0_DB_26"
         ( IN := TRUE,
           PT := #t5,
           Q  := #HOFT,
           ET := #et5
         );


         A     #HOFT;
         JC    SetHOFAlarm;
         JU    BrakefailureAlarm;
   SetHOFAlarm:SET;
         S     "OilFlowHighAlarm";
         S     "OilFlowHighNotify";
         JU    BrakefailureAlarm;
   ResetHOFAlarm:R     "OilFlowHighAlarm";
         R     "OilFlowHighNotify";
         JU    BrakefailureAlarm;
   ResetHOFNotify:R     "OilFlowHighNotify";
         JU    BrakefailureAlarm;
   //-----------------------------------------------------------------------------
   BrakefailureAlarm:L     "RPM";
         L     0;
         >I;
         A     "Brake_Out";
         AN    "AlarmReset";
         AN    "BrakeFailureAlarm";
         JC    BFTimer;
         CALL  RESET_TIMER
         ( "TIMER" := "IEC_Timer_0_DB_27"
         );

         CLR;
         A     "BrakeFailureAlarm";
         A     "AlarmReset";
         FP    #ONS14;
         JC    ResetBFAlarm;
         CLR;
         A     "BrakeFailureNotify";
         A     "AlarmSilence";
         FP    #ONS15;
         JC    ResetBFNotify;
         JU    EstopAlarm;

   BFTimer:CALL  "time conversion"
         ( timein   := "BrakeFailureDelaySpt",
           time_out := #t6
         );
         CALL  TON, "IEC_Timer_0_DB_27"
         ( IN := TRUE,
           PT := #t6,
           Q  := #BFT,
           ET := #et6
         );



         A     #BFT;
         JC    SetBFAlarm;
         JU    EstopAlarm;
   SetBFAlarm:SET;
         S     "BrakeFailureAlarm";
         S     "BrakeFailureNotify";
         JU    EstopAlarm;
   ResetBFAlarm:R     "BrakeFailureAlarm";
         R     "BrakeFailureNotify";
         JU    EstopAlarm;
   ResetBFNotify:R     "BrakeFailureNotify";
         JU    EstopAlarm;
   //-----------------------------------------------------------------------------------
   EstopAlarm:A     "Estop";
         AN    "AlarmReset";
         AN    "EstopAlarm";
         FP    #ONS16;
         JC    SetEAlarm;
         CLR;
         A     "EstopAlarm";
         A     "AlarmReset";
         FP    #ONS17;
         JC    ResetEAlarm;
         CLR;
         A     "EstopNotify";
         A     "AlarmSilence";
         FP    #ONS18;
         JC    ResetENotify;
         BE;

   SetEAlarm:SET;
         S     "EstopAlarm";
         S     "EstopNotify";
         JU    AlarmHorn;
   ResetEAlarm:R     "EstopAlarm";
         R     "EstopNotify";
         JU    AlarmHorn;
   ResetENotify:R     "EstopNotify";
         JU    AlarmHorn;

   //---------------------------------------------------

   AlarmHorn:A     "FaultMode";
         FP    #OS1;
         JC    SetAlarmHorn;
         CLR;
         A     "AlarmReset";
         FP    #OS2;
         JC    ResetAlarmHorn;
         CLR;
         A     "AlarmSilence";
         FP    #OS3;
         JC    ResetAlarmHorn;
         BE;

   SetAlarmHorn:SET;
         S     "Alarm_Horn_Ctrl";
         BE;
   ResetAlarmHorn:SET;
         R     "Alarm_Horn_Ctrl";
         BE;
END_REGION
END_FUNCTION_BLOCK

FUNCTION_BLOCK "HOA_LAD"   // FB10, LAD
{ S7_Optimized_Access := 'TRUE' }
VERSION : 0.1
   VAR
      ONS4 : Bool;
      ONS5 : Bool;
      ONS6 : Bool;
      ONS7 : Bool;
      ONS8 : Bool;
      ONS9 : Bool;
      ONS10 : Bool;
      ONS11 : Bool;
      ONS12 : Bool;
      ONS13 : Bool;
      ONS14 : Bool;
      ONS15 : Bool;
   END_VAR
   VAR_TEMP   // added for the SCL form of the ladder/FBD networks
      _w1 : Bool;
      _w2 : Bool;
      _w3 : Bool;
   END_VAR
BEGIN

REGION Network 1
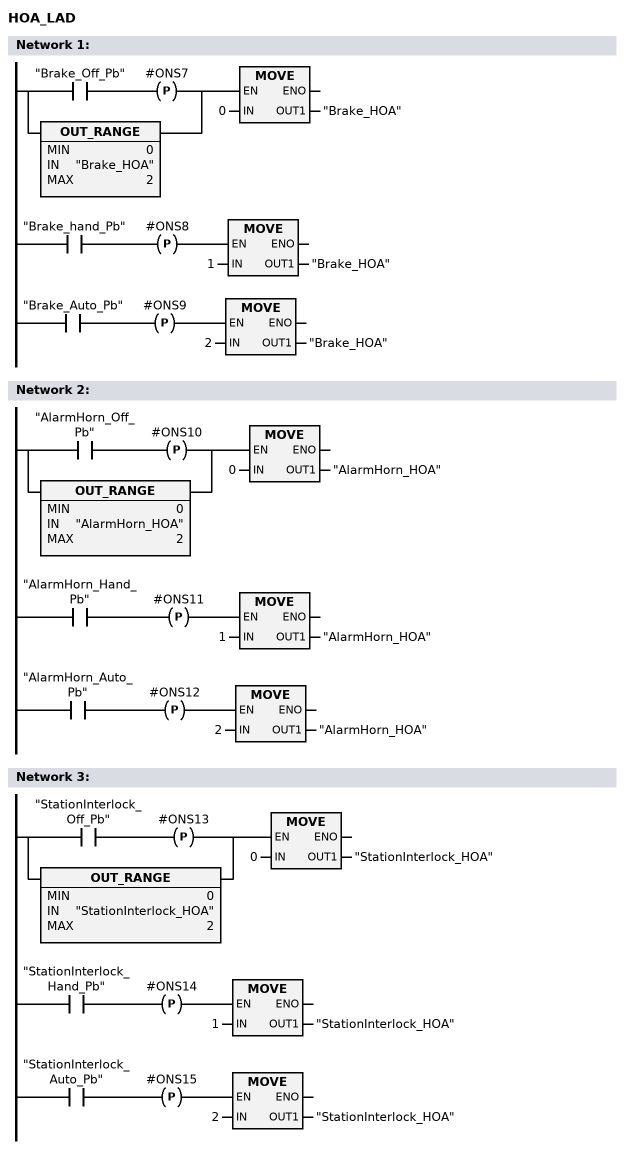
   #_w1 := "Brake_Off_Pb" AND NOT #ONS7;   // rising edge
   #ONS7 := "Brake_Off_Pb";
   IF #_w1 OR ("Brake_HOA" < 0) OR ("Brake_HOA" > 2) THEN "Brake_HOA" := 0; END_IF;
   #_w2 := "Brake_hand_Pb" AND NOT #ONS8;   // rising edge
   #ONS8 := "Brake_hand_Pb";
   IF #_w2 THEN "Brake_HOA" := 1; END_IF;
   #_w3 := "Brake_Auto_Pb" AND NOT #ONS9;   // rising edge
   #ONS9 := "Brake_Auto_Pb";
   IF #_w3 THEN "Brake_HOA" := 2; END_IF;
END_REGION

REGION Network 2
   #_w1 := "AlarmHorn_Off_Pb" AND NOT #ONS10;   // rising edge
   #ONS10 := "AlarmHorn_Off_Pb";
   IF #_w1 OR ("AlarmHorn_HOA" < 0) OR ("AlarmHorn_HOA" > 2) THEN "AlarmHorn_HOA" := 0; END_IF;
   #_w2 := "AlarmHorn_Hand_Pb" AND NOT #ONS11;   // rising edge
   #ONS11 := "AlarmHorn_Hand_Pb";
   IF #_w2 THEN "AlarmHorn_HOA" := 1; END_IF;
   #_w3 := "AlarmHorn_Auto_Pb" AND NOT #ONS12;   // rising edge
   #ONS12 := "AlarmHorn_Auto_Pb";
   IF #_w3 THEN "AlarmHorn_HOA" := 2; END_IF;
END_REGION

REGION Network 3
   #_w1 := "StationInterlock_Off_Pb" AND NOT #ONS13;   // rising edge
   #ONS13 := "StationInterlock_Off_Pb";
   IF #_w1 OR ("StationInterlock_HOA" < 0) OR ("StationInterlock_HOA" > 2) THEN
       "StationInterlock_HOA" := 0;
   END_IF;
   #_w2 := "StationInterlock_Hand_Pb" AND NOT #ONS14;   // rising edge
   #ONS14 := "StationInterlock_Hand_Pb";
   IF #_w2 THEN "StationInterlock_HOA" := 1; END_IF;
   #_w3 := "StationInterlock_Auto_Pb" AND NOT #ONS15;   // rising edge
   #ONS15 := "StationInterlock_Auto_Pb";
   IF #_w3 THEN "StationInterlock_HOA" := 2; END_IF;
END_REGION
END_FUNCTION_BLOCK

FUNCTION_BLOCK "HOA_FBD"   // FB11, FBD
{ S7_Optimized_Access := 'TRUE' }
VERSION : 0.1
   VAR
      ONS4 : Bool;
      ONS5 : Bool;
      ONS6 : Bool;
      ONS7 : Bool;
      ONS8 : Bool;
      ONS9 : Bool;
      ONS10 : Bool;
      ONS11 : Bool;
      ONS12 : Bool;
      ONS13 : Bool;
      ONS14 : Bool;
      ONS15 : Bool;
   END_VAR
   VAR_TEMP   // added for the SCL form of the ladder/FBD networks
      _w1 : Bool;
      _w2 : Bool;
      _w3 : Bool;
   END_VAR
BEGIN

REGION Network 1
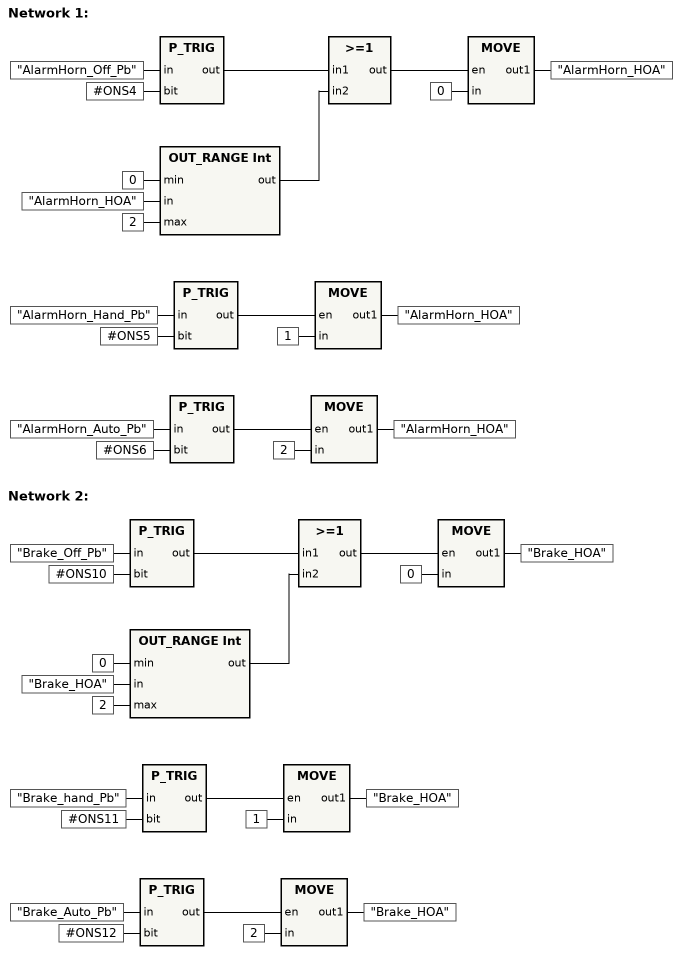
   #_w1 := "AlarmHorn_Off_Pb" AND NOT #ONS4;   // rising edge
   #ONS4 := "AlarmHorn_Off_Pb";
   IF #_w1 OR ("AlarmHorn_HOA" < 0) OR ("AlarmHorn_HOA" > 2) THEN "AlarmHorn_HOA" := 0; END_IF;
   #_w2 := "AlarmHorn_Hand_Pb" AND NOT #ONS5;   // rising edge
   #ONS5 := "AlarmHorn_Hand_Pb";
   IF #_w2 THEN "AlarmHorn_HOA" := 1; END_IF;
   #_w3 := "AlarmHorn_Auto_Pb" AND NOT #ONS6;   // rising edge
   #ONS6 := "AlarmHorn_Auto_Pb";
   IF #_w3 THEN "AlarmHorn_HOA" := 2; END_IF;
END_REGION

REGION Network 2
   #_w1 := "Brake_Off_Pb" AND NOT #ONS10;   // rising edge
   #ONS10 := "Brake_Off_Pb";
   IF #_w1 OR ("Brake_HOA" < 0) OR ("Brake_HOA" > 2) THEN "Brake_HOA" := 0; END_IF;
   #_w2 := "Brake_hand_Pb" AND NOT #ONS11;   // rising edge
   #ONS11 := "Brake_hand_Pb";
   IF #_w2 THEN "Brake_HOA" := 1; END_IF;
   #_w3 := "Brake_Auto_Pb" AND NOT #ONS12;   // rising edge
   #ONS12 := "Brake_Auto_Pb";
   IF #_w3 THEN "Brake_HOA" := 2; END_IF;
END_REGION

REGION Network 3
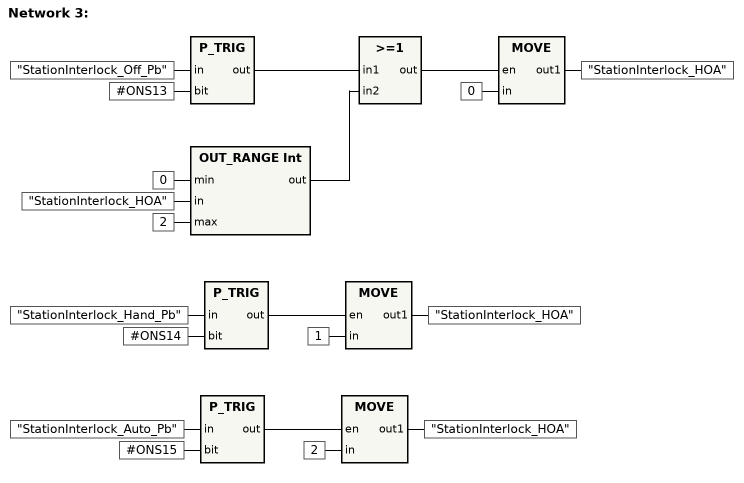
   #_w1 := "StationInterlock_Off_Pb" AND NOT #ONS13;   // rising edge
   #ONS13 := "StationInterlock_Off_Pb";
   IF #_w1 OR ("StationInterlock_HOA" < 0) OR ("StationInterlock_HOA" > 2) THEN
       "StationInterlock_HOA" := 0;
   END_IF;
   #_w2 := "StationInterlock_Hand_Pb" AND NOT #ONS14;   // rising edge
   #ONS14 := "StationInterlock_Hand_Pb";
   IF #_w2 THEN "StationInterlock_HOA" := 1; END_IF;
   #_w3 := "StationInterlock_Auto_Pb" AND NOT #ONS15;   // rising edge
   #ONS15 := "StationInterlock_Auto_Pb";
   IF #_w3 THEN "StationInterlock_HOA" := 2; END_IF;
END_REGION
END_FUNCTION_BLOCK

FUNCTION_BLOCK "HOA_SCL"   // FB12, SCL
{ S7_Optimized_Access := 'TRUE' }
VERSION : 0.1
BEGIN

   //------------------------------------------------------------------------
   //Brake_HOA controls

   IF "Brake_HOA" < 0 OR "Brake_HOA" > 2 THEN
       "Brake_HOA" := 0;
   END_IF;

   IF "Brake_Off_Pb" AND "Brake_HOA" <> 0 THEN
       "Brake_HOA" := 0;
   END_IF;

   IF "Brake_hand_Pb" AND "Brake_HOA" <> 1 THEN
       "Brake_HOA" := 1;
   END_IF;

   IF "Brake_Auto_Pb" AND "Brake_HOA" <> 2 THEN
       "Brake_HOA" := 2;
   END_IF;
   //-----------------------------------------------------------------------------
   //AlarmHorn_HOA controls

   IF "AlarmHorn_HOA" < 0 OR "AlarmHorn_HOA" > 2 THEN
       "AlarmHorn_HOA" := 0;
   END_IF;

   IF "AlarmHorn_Off_Pb" AND "AlarmHorn_HOA" <> 0 THEN
       "AlarmHorn_HOA" := 0;
   END_IF;

   IF "AlarmHorn_Hand_Pb" AND "AlarmHorn_HOA" <> 1 THEN
       "AlarmHorn_HOA" := 1;
   END_IF;

   IF "AlarmHorn_Auto_Pb" AND "AlarmHorn_HOA" <> 2 THEN
       "AlarmHorn_HOA" := 2;
   END_IF;
   //--------------------------------------------------------------------------
   //StationInterlock_HOA controls

   IF "StationInterlock_HOA" < 0 OR "StationInterlock_HOA" > 2 THEN
       "StationInterlock_HOA" := 0;
   END_IF;

   IF "StationInterlock_Off_Pb" AND "StationInterlock_HOA" <> 0 THEN
       "StationInterlock_HOA" := 0;
   END_IF;

   IF "StationInterlock_Hand_Pb" AND "StationInterlock_HOA" <> 1 THEN
       "StationInterlock_HOA" := 1;
   END_IF;

   IF "StationInterlock_Auto_Pb" AND "StationInterlock_HOA" <> 2 THEN
       "StationInterlock_HOA" := 2;
   END_IF;
END_FUNCTION_BLOCK

FUNCTION_BLOCK "HOA_STL"   // FB13, STL
{ S7_Optimized_Access := 'TRUE' }
VERSION : 0.1
   VAR
      ONS4 : Bool;
      ONS5 : Bool;
      ONS6 : Bool;
      ONS7 : Bool;
      ONS8 : Bool;
      ONS9 : Bool;
      ONS10 : Bool;
      ONS11 : Bool;
      ONS12 : Bool;
      ONS13 : Bool;
      ONS14 : Bool;
      ONS15 : Bool;
   END_VAR
BEGIN

REGION Network 1

   //------------------------------------------------

   Brake:L     "Brake_HOA";
         L     0;
         <I;
         JC    SetBrakeZero;
         CLR;
         L     "Brake_HOA";
         L     2;
         >I;
         JC    SetBrakeZero;
         CLR;
         A     "Brake_Off_Pb";
         FP    #ONS7;
         JC    SetBrakeZero;
         CLR;
         A     "Brake_hand_Pb";
         FP    #ONS8;
         JC    SetBrakeOne;
         CLR;
         A     "Brake_Auto_Pb";
         FP    #ONS9;
         JC    SetBrakeTwo;
         JU    AlarmHorn;



   SetBrakeZero:L     0;
         T     "Brake_HOA";
         JU    AlarmHorn;
   SetBrakeOne:L     1;
         T     "Brake_HOA";
         JC    AlarmHorn;
   SetBrakeTwo:L     2;
         T     "Brake_HOA";
         JU    AlarmHorn;

   //-------------------------------------------------------------
   AlarmHorn:L     "AlarmHorn_HOA";
         L     0;
         <I;
         JC    SetAlarmHornZero;
         CLR;
         L     "AlarmHorn_HOA";
         L     2;
         >I;
         JC    SetBrakeZero;
         CLR;
         A     "AlarmHorn_Off_Pb";
         FP    #ONS10;
         JC    SetAlarmHornZero;
         CLR;
         A     "AlarmHorn_Hand_Pb";
         FP    #ONS11;
         JC    SetAlarmHornOne;
         CLR;
         A     "AlarmHorn_Auto_Pb";
         FP    #ONS12;
         JC    SetAlarmHornTwo;
         JU    Interlock;



   SetAlarmHornZero:L     0;
         T     "Brake_HOA";
         JU    Interlock;
   SetAlarmHornOne:L     1;
         T     "Brake_HOA";
         JC    Interlock;
   SetAlarmHornTwo:L     2;
         T     "Brake_HOA";
         JU    Interlock;

   //--------------------------------------------------------------

   Interlock:L     "StationInterlock_HOA";
         L     0;
         <I;
         JC    SetStationZero;
         CLR;
         L     "StationInterlock_HOA";
         L     2;
         >I;
         JC    SetStationZero;
         CLR;
         A     "StationInterlock_Off_Pb";
         FP    #ONS13;
         JC    SetAlarmHornZero;
         CLR;
         A     "StationInterlock_Auto_Pb";
         FP    #ONS14;
         JC    SetStationOne;
         CLR;
         A     "StationInterlock_Auto_Pb";
         FP    #ONS15;
         JC    SetStationTwo;
         JU    EndOfLine;



   SetStationZero:L     0;
         T     "StationInterlock_HOA";
         BE;
   SetStationOne:L     1;
         T     "StationInterlock_HOA";
         BE;
   SetStationTwo:L     2;
         T     "StationInterlock_HOA";
         BE;
   EndOfLine:BE;
END_REGION
END_FUNCTION_BLOCK

FUNCTION_BLOCK "MODES_LAD"   // FB14, LAD
{ S7_Optimized_Access := 'TRUE' }
VERSION : 0.1
   VAR
      et1 : Time;
      ONS4 : Bool;
      ONS5 : Bool;
      ONS6 : Bool;
      ONS7 : Bool;
      ONS8 : Bool;
   END_VAR
   VAR_TEMP
      tv1 : Time;
      v1 : Int;
      v2 : Int;
      et2 : Time;
      tv2 : Time;
      tv3 : Time;
      et3 : Time;
   END_VAR
   VAR_TEMP   // added for the SCL form of the ladder/FBD networks
      _w1 : Bool;
      _w2 : Bool;
      _w3 : Bool;
   END_VAR
BEGIN

REGION Network 1
   // Warmup mode:
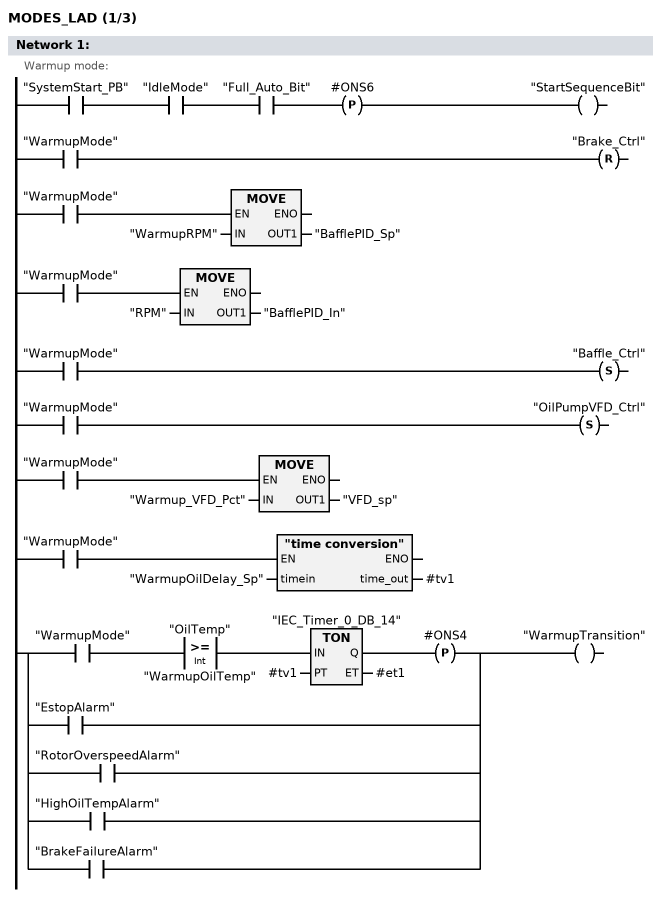
   #_w1 := "SystemStart_PB" AND "IdleMode" AND "Full_Auto_Bit";
   #_w2 := #_w1 AND NOT #ONS6;   // rising edge
   #ONS6 := #_w1;
   "StartSequenceBit" := #_w2;
   IF "WarmupMode" THEN
       "Brake_Ctrl" := FALSE;
       "BafflePID_Sp" := "WarmupRPM";
       "BafflePID_In" := "RPM";
       "Baffle_Ctrl" := TRUE;
       "OilPumpVFD_Ctrl" := TRUE;
       "VFD_sp" := "Warmup_VFD_Pct";
       "time conversion"(timein := "WarmupOilDelay_Sp", time_out => #tv1);
   END_IF;
   "IEC_Timer_0_DB_14".TON(IN := "WarmupMode" AND ("OilTemp" >= "WarmupOilTemp"), PT := #tv1, ET => #et1);
   #_w3 := "IEC_Timer_0_DB_14".Q AND NOT #ONS4;   // rising edge
   #ONS4 := "IEC_Timer_0_DB_14".Q;
   "WarmupTransition" := #_w3 OR "EstopAlarm" OR "RotorOverspeedAlarm" OR "HighOilTempAlarm" OR "BrakeFailureAlarm";
END_REGION

REGION Network 2
   // Stabilize Mode:
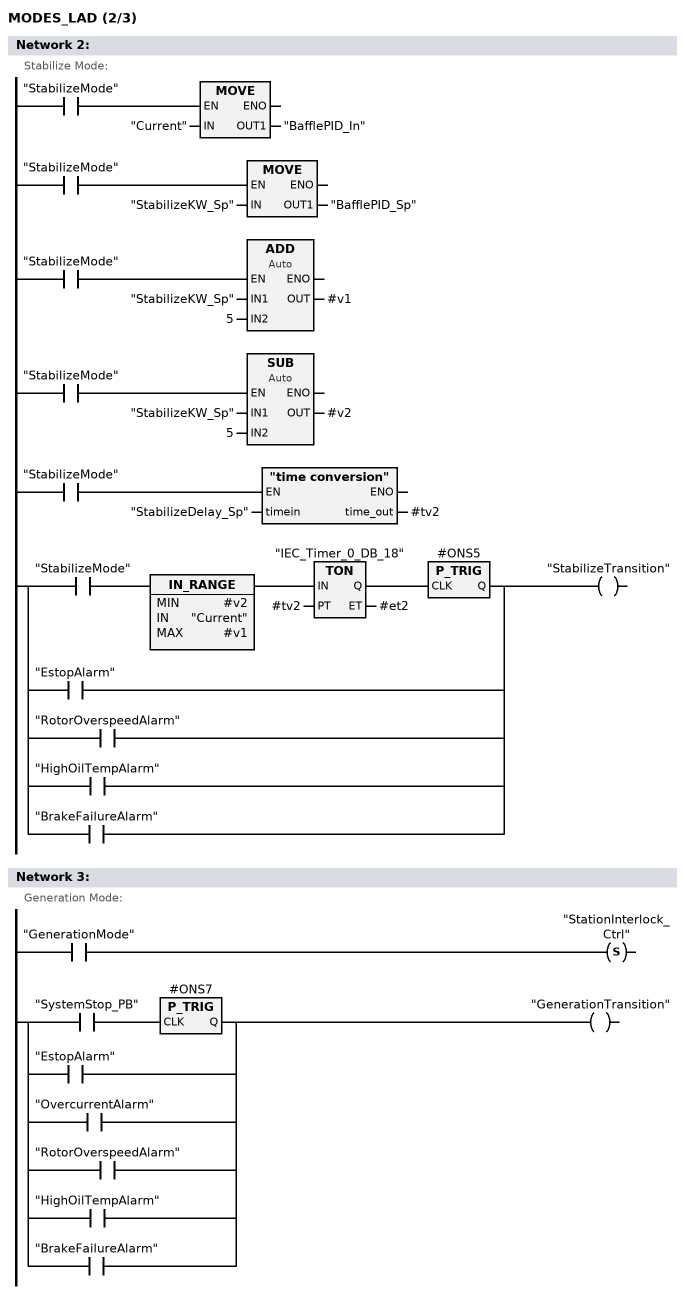
   IF "StabilizeMode" THEN
       "BafflePID_In" := "Current";
       "BafflePID_Sp" := "StabilizeKW_Sp";
       #v1 := "StabilizeKW_Sp" + 5;
       #v2 := "StabilizeKW_Sp" - 5;
       "time conversion"(timein := "StabilizeDelay_Sp", time_out => #tv2);
   END_IF;
   "IEC_Timer_0_DB_18".TON(IN := "StabilizeMode" AND (#v2 <= "Current") AND ("Current" <= #v1),
                           PT := #tv2,
                           ET => #et2);
   #_w1 := "IEC_Timer_0_DB_18".Q AND NOT #ONS5;   // rising edge
   #ONS5 := "IEC_Timer_0_DB_18".Q;
   "StabilizeTransition" := #_w1 OR "EstopAlarm" OR "RotorOverspeedAlarm" OR "HighOilTempAlarm" OR "BrakeFailureAlarm";
END_REGION

REGION Network 3
   // Generation Mode:
   RUNG wire#powerrail
      Contact( "GenerationMode" )
      S_Coil( "StationInterlock_Ctrl" )
   END_RUNG
   RUNG wire#powerrail
      Contact( "SystemStop_PB" )
      P_Trig( #ONS7 )
      wire#w1
      Coil( "GenerationTransition" )
   END_RUNG
   RUNG wire#powerrail
      Contact( "EstopAlarm" )
   END_RUNG wire#w1
   RUNG wire#powerrail
      Contact( "OvercurrentAlarm" )
   END_RUNG wire#w1
   RUNG wire#powerrail
      Contact( "RotorOverspeedAlarm" )
   END_RUNG wire#w1
   RUNG wire#powerrail
      Contact( "HighOilTempAlarm" )
   END_RUNG wire#w1
   RUNG wire#powerrail
      Contact( "BrakeFailureAlarm" )
   END_RUNG wire#w1
   // the same network as SCL:
   IF "GenerationMode" THEN "StationInterlock_Ctrl" := TRUE; END_IF;
   #_w1 := "SystemStop_PB" AND NOT #ONS7;   // rising edge
   #ONS7 := "SystemStop_PB";
   "GenerationTransition" := #_w1 OR "EstopAlarm" OR "OvercurrentAlarm" OR "RotorOverspeedAlarm" OR "HighOilTempAlarm" OR "BrakeFailureAlarm";
END_REGION

REGION Network 4
   // Cooldown Mode:
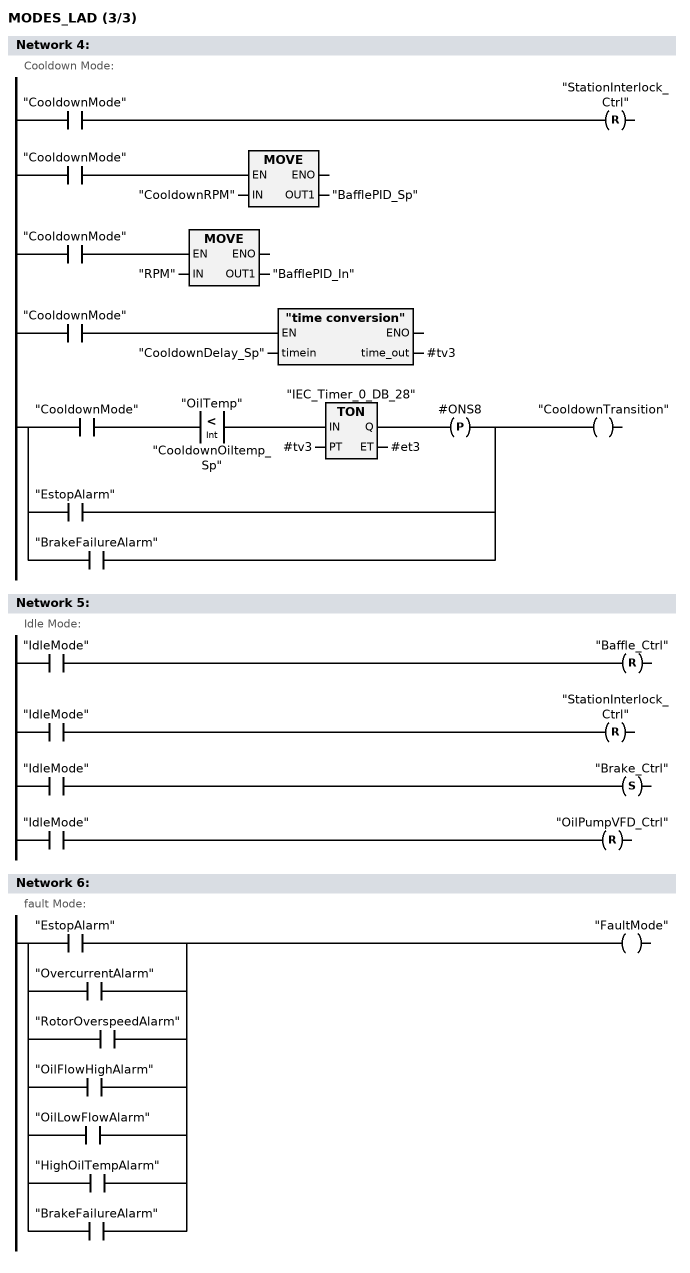
   IF "CooldownMode" THEN
       "StationInterlock_Ctrl" := FALSE;
       "BafflePID_Sp" := "CooldownRPM";
       "BafflePID_In" := "RPM";
       "time conversion"(timein := "CooldownDelay_Sp", time_out => #tv3);
   END_IF;
   "IEC_Timer_0_DB_28".TON(IN := "CooldownMode" AND ("OilTemp" < "CooldownOiltemp_Sp"), PT := #tv3, ET => #et3);
   #_w1 := "IEC_Timer_0_DB_28".Q AND NOT #ONS8;   // rising edge
   #ONS8 := "IEC_Timer_0_DB_28".Q;
   "CooldownTransition" := #_w1 OR "EstopAlarm" OR "BrakeFailureAlarm";
END_REGION

REGION Network 5
   // Idle Mode:
   RUNG wire#powerrail
      Contact( "IdleMode" )
      R_Coil( "Baffle_Ctrl" )
   END_RUNG
   RUNG wire#powerrail
      Contact( "IdleMode" )
      R_Coil( "StationInterlock_Ctrl" )
   END_RUNG
   RUNG wire#powerrail
      Contact( "IdleMode" )
      S_Coil( "Brake_Ctrl" )
   END_RUNG
   RUNG wire#powerrail
      Contact( "IdleMode" )
      R_Coil( "OilPumpVFD_Ctrl" )
   END_RUNG
   // the same network as SCL:
   IF "IdleMode" THEN
       "Baffle_Ctrl" := FALSE;
       "StationInterlock_Ctrl" := FALSE;
       "Brake_Ctrl" := TRUE;
       "OilPumpVFD_Ctrl" := FALSE;
   END_IF;
END_REGION

REGION Network 6
   // fault Mode:
   RUNG wire#powerrail
      Contact( "EstopAlarm" )
      wire#w1
      Coil( "FaultMode" )
   END_RUNG
   RUNG wire#powerrail
      Contact( "OvercurrentAlarm" )
   END_RUNG wire#w1
   RUNG wire#powerrail
      Contact( "RotorOverspeedAlarm" )
   END_RUNG wire#w1
   RUNG wire#powerrail
      Contact( "OilFlowHighAlarm" )
   END_RUNG wire#w1
   RUNG wire#powerrail
      Contact( "OilLowFlowAlarm" )
   END_RUNG wire#w1
   RUNG wire#powerrail
      Contact( "HighOilTempAlarm" )
   END_RUNG wire#w1
   RUNG wire#powerrail
      Contact( "BrakeFailureAlarm" )
   END_RUNG wire#w1
   // the same network as SCL:
   "FaultMode" := "EstopAlarm" OR "OvercurrentAlarm" OR "RotorOverspeedAlarm" OR "OilFlowHighAlarm" OR "OilLowFlowAlarm" OR "HighOilTempAlarm" OR "BrakeFailureAlarm";
END_REGION
END_FUNCTION_BLOCK

FUNCTION_BLOCK "MODES_FBD"   // FB15, FBD
{ S7_Optimized_Access := 'TRUE' }
VERSION : 0.1
   VAR
      ONS4 : Bool;
      ONS5 : Bool;
      ONS6 : Bool;
      ONS7 : Bool;
      ONS8 : Bool;
   END_VAR
   VAR_TEMP
      tv1 : Time;
      et1 : Time;
      v1 : Int;
      v2 : Int;
      tv2 : Time;
      et2 : Time;
      tv3 : Time;
      et3 : Time;
   END_VAR
   VAR_TEMP   // added for the SCL form of the ladder/FBD networks
      _w1 : Bool;
      _w2 : Bool;
      _w3 : Bool;
   END_VAR
BEGIN

REGION Network 1
   // Warmup Mode
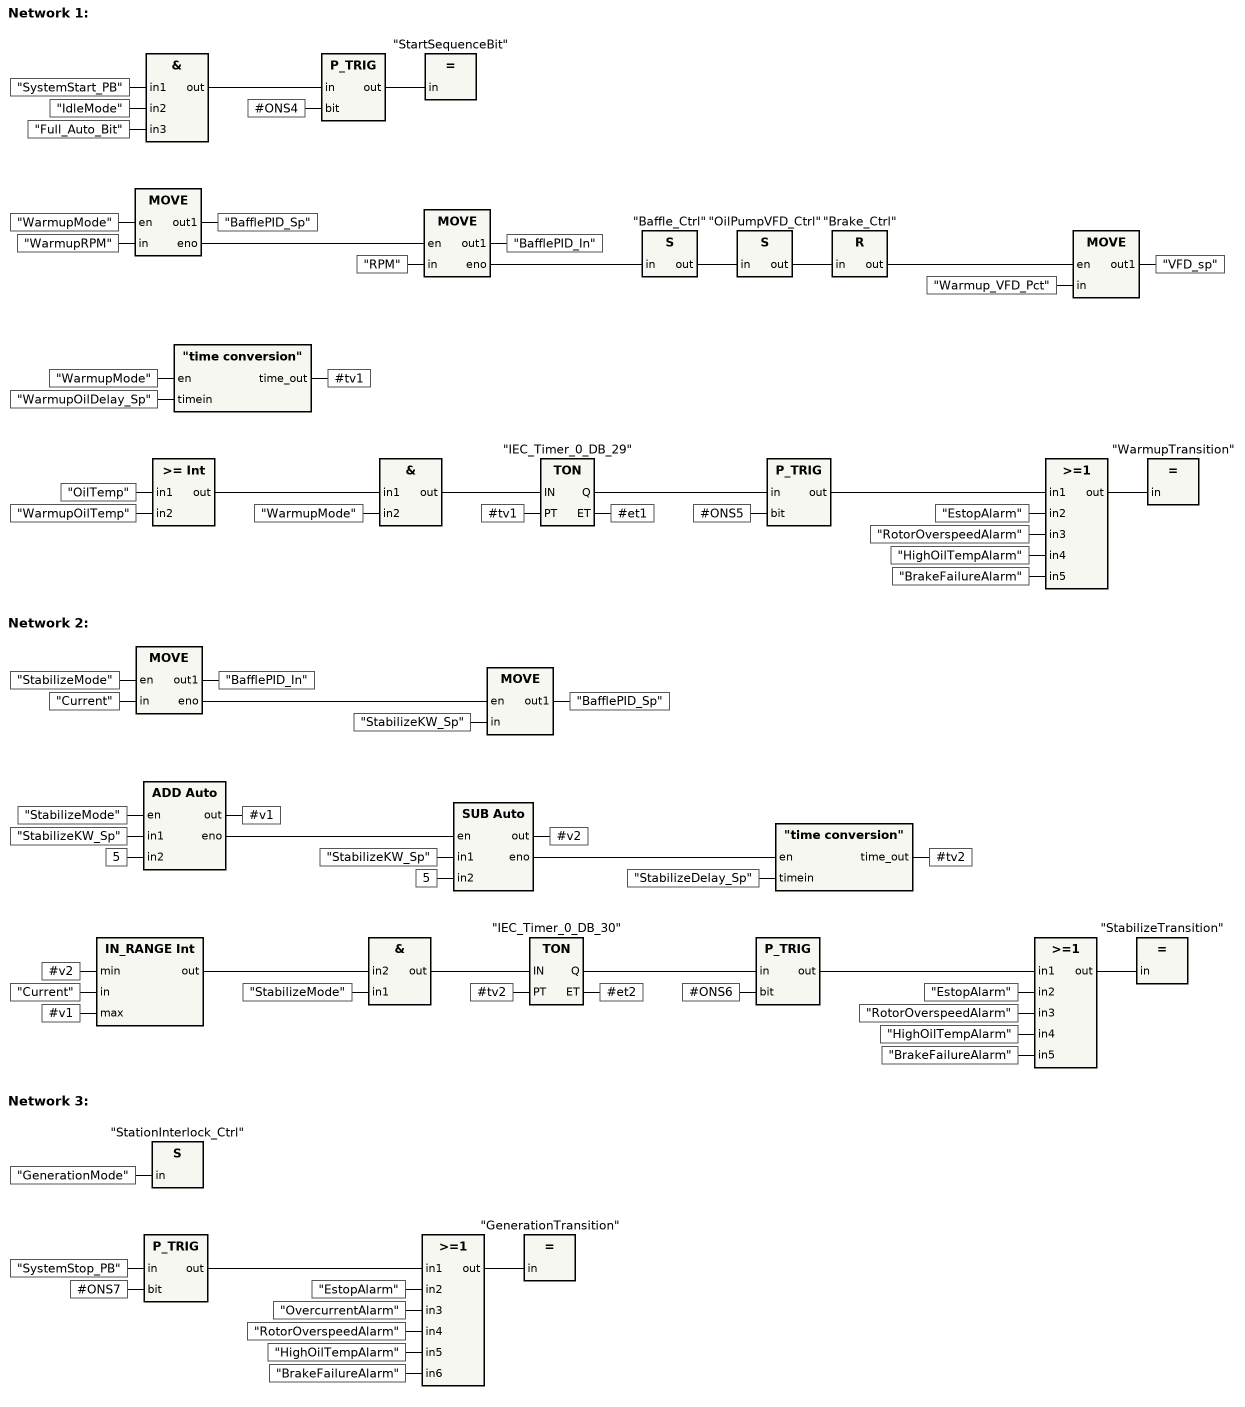
   #_w1 := "SystemStart_PB" AND "IdleMode" AND "Full_Auto_Bit";
   #_w2 := #_w1 AND NOT #ONS4;   // rising edge
   #ONS4 := #_w1;
   "StartSequenceBit" := #_w2;
   IF "WarmupMode" THEN
       "BafflePID_Sp" := "WarmupRPM";
       "BafflePID_In" := "RPM";
       "Baffle_Ctrl" := TRUE;
       "OilPumpVFD_Ctrl" := TRUE;
       "Brake_Ctrl" := FALSE;
       "VFD_sp" := "Warmup_VFD_Pct";
       "time conversion"(timein := "WarmupOilDelay_Sp", time_out => #tv1);
   END_IF;
   "IEC_Timer_0_DB_29".TON(IN := ("OilTemp" >= "WarmupOilTemp") AND "WarmupMode", PT := #tv1, ET => #et1);
   #_w3 := "IEC_Timer_0_DB_29".Q AND NOT #ONS5;   // rising edge
   #ONS5 := "IEC_Timer_0_DB_29".Q;
   "WarmupTransition" := #_w3 OR "EstopAlarm" OR "RotorOverspeedAlarm" OR "HighOilTempAlarm" OR "BrakeFailureAlarm";
END_REGION

REGION Network 2
   // Stabilize Mode:
   IF "StabilizeMode" THEN
       "BafflePID_In" := "Current";
       "BafflePID_Sp" := "StabilizeKW_Sp";
       #v1 := "StabilizeKW_Sp" + 5;
       #v2 := "StabilizeKW_Sp" - 5;
       "time conversion"(timein := "StabilizeDelay_Sp", time_out => #tv2);
   END_IF;
   "IEC_Timer_0_DB_30".TON(IN := (#v2 <= "Current") AND ("Current" <= #v1) AND "StabilizeMode",
                           PT := #tv2,
                           ET => #et2);
   #_w1 := "IEC_Timer_0_DB_30".Q AND NOT #ONS6;   // rising edge
   #ONS6 := "IEC_Timer_0_DB_30".Q;
   "StabilizeTransition" := #_w1 OR "EstopAlarm" OR "RotorOverspeedAlarm" OR "HighOilTempAlarm" OR "BrakeFailureAlarm";
END_REGION

REGION Network 3
   // Generation Mode:
   IF "GenerationMode" THEN "StationInterlock_Ctrl" := TRUE; END_IF;
   #_w1 := "SystemStop_PB" AND NOT #ONS7;   // rising edge
   #ONS7 := "SystemStop_PB";
   "GenerationTransition" := #_w1 OR "EstopAlarm" OR "OvercurrentAlarm" OR "RotorOverspeedAlarm" OR "HighOilTempAlarm" OR "BrakeFailureAlarm";
END_REGION

REGION Network 4
   // CooldownMode:
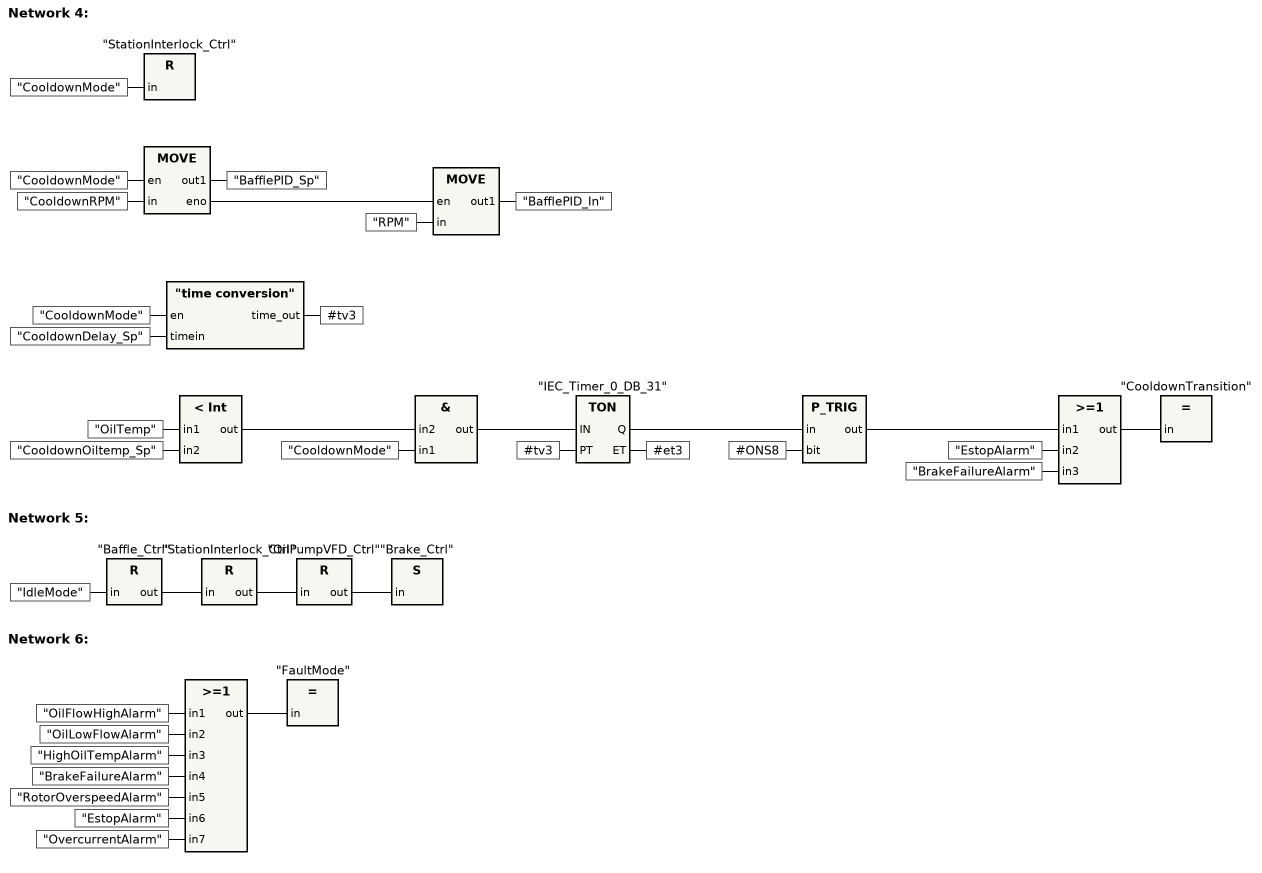
   IF "CooldownMode" THEN
       "StationInterlock_Ctrl" := FALSE;
       "BafflePID_Sp" := "CooldownRPM";
       "BafflePID_In" := "RPM";
       "time conversion"(timein := "CooldownDelay_Sp", time_out => #tv3);
   END_IF;
   "IEC_Timer_0_DB_31".TON(IN := ("OilTemp" < "CooldownOiltemp_Sp") AND "CooldownMode", PT := #tv3, ET => #et3);
   #_w1 := "IEC_Timer_0_DB_31".Q AND NOT #ONS8;   // rising edge
   #ONS8 := "IEC_Timer_0_DB_31".Q;
   "CooldownTransition" := #_w1 OR "EstopAlarm" OR "BrakeFailureAlarm";
END_REGION

REGION Network 5
   // Idle Mode:
   IF "IdleMode" THEN
       "Baffle_Ctrl" := FALSE;
       "StationInterlock_Ctrl" := FALSE;
       "OilPumpVFD_Ctrl" := FALSE;
       "Brake_Ctrl" := TRUE;
   END_IF;
END_REGION

REGION Network 6
   // fault Mode:
   "FaultMode" := "OilFlowHighAlarm" OR "OilLowFlowAlarm" OR "HighOilTempAlarm" OR "BrakeFailureAlarm" OR "RotorOverspeedAlarm" OR "EstopAlarm" OR "OvercurrentAlarm";
END_REGION
END_FUNCTION_BLOCK

FUNCTION_BLOCK "MODES_SCL"   // FB16, SCL
{ S7_Optimized_Access := 'TRUE' }
VERSION : 0.1
   VAR_TEMP
      tv1 : Time;
      et1 : Time;
      tv2 : Time;
      et2 : Time;
      warmupTrigger : Bool;
      stablizeTrigger : Bool;
      tv3 : Time;
      et3 : Time;
      CooldownTrigger : Bool;
   END_VAR
BEGIN
   //Estop Alarm:
   IF "EstopAlarm"OR "BrakeFailureAlarm" THEN
       "WarmupTransition" := 1;
       "StabilizeTransition" := 1;
       "GenerationTransition" := 1;
       "CooldownTransition" := 1;

   ELSE

       //Warmup Mode:
       IF "SystemStart_PB" AND "IdleMode" AND "Full_Auto_Bit" THEN
           "StartSequenceBit" := 1;
       ELSE
           "StartSequenceBit" := 0;
       END_IF;
       IF "WarmupMode" THEN
           "BafflePID_In" := "RPM";
           "BafflePID_Sp" := "WarmupRPM";
           "Baffle_Ctrl" := 1;
           "Brake_Ctrl" := 0;
           "OilPumpVFD_Ctrl" := 1;
           "VFD_sp" := "Warmup_VFD_Pct";
           IF "OilTemp" >= "WarmupOilTemp" THEN
               "time conversion"(timein := "WarmupOilDelay_Sp",
                                 time_out => #tv1);

               "IEC_Timer_0_DB_32".TON(IN := TRUE,
                                       PT := #tv1,
                                       Q => #warmupTrigger,
                                       ET => #et1);
           ELSE
               RESET_TIMER("IEC_Timer_0_DB_32");
           END_IF;
           IF #warmupTrigger THEN
               RESET_TIMER("IEC_Timer_0_DB_32");

               "WarmupTransition" := 1;
           END_IF;
       ELSE
           "WarmupTransition" := 0;

       END_IF;
       IF "RotorOverspeedAlarm" OR "HighOilTempAlarm" THEN
           "WarmupTransition" := 1;
       END_IF;


       //Stabilize Mode
       IF "StabilizeMode" THEN
           "BafflePID_In" := "Current";
           "BafflePID_Sp" := "StabilizeKW_Sp";

           IF "Current" < ("StabilizeKW_Sp" + 5) AND "Current" > ("StabilizeKW_Sp" - 5) THEN
               "time conversion"(timein := "StabilizeDelay_Sp",
                                 time_out => #tv2);

               "IEC_Timer_0_DB_33".TON(IN := TRUE,
                                       PT := #tv2,
                                       Q => #stablizeTrigger,
                                       ET => #et2);
           ELSE
               RESET_TIMER("IEC_Timer_0_DB_33");
           END_IF;
           IF #stablizeTrigger THEN
               RESET_TIMER("IEC_Timer_0_DB_33");
               "StabilizeTransition" := 1;
           END_IF;
           ;
       ELSE
           "StabilizeTransition" := 0;
       END_IF;
       IF "RotorOverspeedAlarm"OR "HighOilTempAlarm" THEN
           "StabilizeTransition" := 1;
       END_IF;


       //Generation mode

       IF "GenerationMode" AND NOT "OvercurrentAlarm" THEN
           "StationInterlock_Ctrl" := 1;
           IF "SystemStop_PB" THEN
               "GenerationTransition" := 1;
           END_IF;
       ELSE
           "GenerationTransition" := 0;
       END_IF;
       IF "OvercurrentAlarm" OR "RotorOverspeedAlarm" OR "HighOilTempAlarm" THEN
           "GenerationTransition" := 1;
       END_IF;


       //Cooldown Mode
       IF "CooldownMode" THEN
           "StationInterlock_Ctrl" := 0;
           "BafflePID_In" := "RPM";
           "BafflePID_Sp" := "CooldownRPM";

           IF "OilTemp" < "CooldownOiltemp_Sp" THEN
               "time conversion"(timein := "CooldownDelay_Sp",
                                 time_out => #tv3);
               "IEC_Timer_0_DB_34".TON(IN := TRUE,
                                       PT := #tv3,
                                       Q => #CooldownTrigger,
                                       ET => #et3);
           ELSE
               RESET_TIMER("IEC_Timer_0_DB_34");
           END_IF;
           IF #CooldownTrigger THEN
               RESET_TIMER("IEC_Timer_0_DB_34");
               "CooldownTransition" := 1;
           END_IF;

       ELSE
           "CooldownTransition" := 0;
       END_IF;


       //Fault Mode
       IF "EstopAlarm" OR "OvercurrentAlarm" OR "RotorOverspeedAlarm" OR "HighOilTempAlarm" OR "OilFlowHighAlarm" OR "OilLowFlowAlarm" OR "BrakeFailureAlarm" THEN
           "FaultMode" := 1;
       ELSE
           "FaultMode" := 0;
       END_IF;
   END_IF;

   //Idle mode
   IF "IdleMode" THEN
       "Baffle_Ctrl" := 0;
       "StationInterlock_Ctrl" := 0;
       "OilPumpVFD_Ctrl" := 0;
       "Brake_Ctrl" := 1;
   ELSE
       "IdleMode" := 0;
   END_IF;
END_FUNCTION_BLOCK

FUNCTION_BLOCK "MODES_STL"   // FB17, STL
{ S7_Optimized_Access := 'TRUE' }
VERSION : 0.1
   VAR
      ONS4 : Bool;
      ONS5 : Bool;
   END_VAR
   VAR_TEMP
      tv1 : Time;
      warmupTrigger : Bool;
      et1 : Time;
      v1 : Int;
      v2 : Int;
      tb1 : Bool;
      tv2 : Time;
      stabilizetrigger : Bool;
      et2 : Time;
      tv3 : Time;
      cooldowntrigger : Bool;
      et3 : Time;
   END_VAR
BEGIN

REGION Network 1
   //EStop handler
   Estop:A     "EstopAlarm";
         O     "BrakeFailureAlarm";
         JC    Estoptransitions;
         JU    Startwarmup;
   Estoptransitions:SET;
         S     "WarmupTransition";
         S     "StabilizeTransition";
         S     "GenerationTransition";
         S     "CooldownTransition";
         JU    IdleMode;
   Startwarmup:SET;
         R     "WarmupTransition";
         R     "StabilizeTransition";
         R     "GenerationTransition";
         R     "CooldownTransition";

         A     "SystemStart_PB";
         FP    #ONS4;
         A     "IdleMode";
         A     "Full_Auto_Bit";
         S     "StartSequenceBit";
         CLR;

   //Warmup mode
   WarmupMode:AN    "WarmupMode";
         A     "StartSequenceBit";
         JC    stabilizeMode;
         SET;

         R     "Brake_Ctrl";
         R     "StartSequenceBit";
         L     "WarmupRPM";
         T     "BafflePID_Sp";
         L     "RPM";
         T     "BafflePID_In";
         L     "Warmup_VFD_Pct";
         T     "VFD_sp";
         SET;
         S     "OilPumpVFD_Ctrl";
         S     "Baffle_Ctrl";
         L     "OilTemp";
         L     "WarmupOilTemp";
         >=I;
         JC    warmuptime;
         CALL  RESET_TIMER
         ( "TIMER" := "IEC_Timer_0_DB_35"
         );

         JU    stabilizeMode;
   warmuptime:CALL  "time conversion"
         ( timein   := "WarmupOilDelay_Sp",
           time_out := #tv1
         );
         CALL  TON, "IEC_Timer_0_DB_35"
         ( IN := TRUE,
           PT := #tv1,
           Q  := #warmupTrigger,
           ET := #et1
         );

         A     #warmupTrigger;
         JC    warmupExit;
         CLR;
         A     "RotorOverspeedAlarm";
         JC    warmupExit;
         CLR;
         A     "HighOilTempAlarm";
         JC    warmupExit;
         JU    stabilizeMode;

   warmupExit:S     "WarmupTransition";
         CALL  RESET_TIMER
         ( "TIMER" := "IEC_Timer_0_DB_35"
         );

   //Stabilize Mode
   stabilizeMode:AN    "StabilizeMode";
         JC    GenerationMode;
         SET;
         R     "WarmupTransition";
         L     "Current";
         T     "BafflePID_In";
         L     "StabilizeKW_Sp";
         T     "BafflePID_Sp";

         L     "StabilizeKW_Sp";
         L     5;
         +I;
         T     #v1;

         L     "StabilizeKW_Sp";
         L     5;
         -I;
         T     #v2;

         L     "Current";
         L     #v1;
         <I;
         S     #tb1;
         L     "Current";
         L     #v2;
         >I;
         A     #tb1;
         JC    stabilizeTime;
         CALL  RESET_TIMER
         ( "TIMER" := "IEC_Timer_0_DB_36"
         );
         JU    GenerationMode;

   stabilizeTime:CALL  "time conversion"
         ( timein   := "StabilizeDelay_Sp",
           time_out := #tv2
         );
         CALL  TON, "IEC_Timer_0_DB_36"
         ( IN := TRUE,
           PT := #tv2,
           Q  := #stabilizetrigger,
           ET := #et2
         );
         A     #stabilizetrigger;
         JC    stabilizeExit;
         CLR;
         A     "RotorOverspeedAlarm";
         JC    stabilizeExit;
         CLR;
         A     "HighOilTempAlarm";
         JC    stabilizeExit;
         JU    GenerationMode;
   stabilizeExit:S     "StabilizeTransition";
         CALL  RESET_TIMER
         ( "TIMER" := "IEC_Timer_0_DB_36"
         );
   //Generation Mode
   GenerationMode:AN    "GenerationMode";
         JC    CoolDownMode;
         SET;
         R     "StabilizeTransition";
         SET;
         S     "StationInterlock_Ctrl";
         CLR;
         A     "SystemStop_PB";
         FP    #ONS5;
         O     "OvercurrentAlarm";
         O     "RotorOverspeedAlarm";
         O     "HighOilTempAlarm";
         S     "GenerationTransition";
   //CoolDown Mode
   CoolDownMode:AN    "CooldownMode";
         JC    IdleMode;
         SET;
         R     "GenerationTransition";
         R     "StationInterlock_Ctrl";
         L     "CooldownRPM";
         T     "BafflePID_Sp";
         L     "RPM";
         T     "BafflePID_In";
         L     "OilTemp";
         L     "CooldownOiltemp_Sp";
         <I;
         JC    cooldownTime;
         CALL  RESET_TIMER
         ( "TIMER" := "IEC_Timer_0_DB_37"
         );


         JU    IdleMode;
   cooldownTime:CALL  "time conversion"
         ( timein   := "CooldownDelay_Sp",
           time_out := #tv3
         );

         CALL  TON, "IEC_Timer_0_DB_37"
         ( IN := TRUE,
           PT := #tv3,
           Q  := #cooldowntrigger,
           ET := #et3
         );
         A     #cooldowntrigger;
         JC    cooldownExit;
         JU    IdleMode;
   cooldownExit:S     "CooldownTransition";
         CALL  RESET_TIMER
         ( "TIMER" := "IEC_Timer_0_DB_37"
         );
   //Idle Mode
   IdleMode:AN    "IdleMode";
         JC    EndOfLine;
         SET;
         R     "CooldownTransition";
         R     "Baffle_Ctrl";
         R     "StationInterlock_Ctrl";
         R     "OilPumpVFD_Ctrl";
         SET;
         S     "Brake_Ctrl";
   //Fault Mode
   EndOfLine:A     "EstopAlarm";
         O     "OilFlowHighAlarm";
         O     "OilLowFlowAlarm";
         O     "HighOilTempAlarm";
         O     "RotorOverspeedAlarm";
         O     "OvercurrentAlarm";
         O     "BrakeFailureAlarm";
         =     "FaultMode";
         BE;
END_REGION
END_FUNCTION_BLOCK

